C09063=1055.892,154.749,-84.853,171.715,33.030,156.169
C09064=1055.897,154.998,-84.876,171.717,33.033,156.169
C09065=1055.904,155.247,-84.898,171.719,33.035,156.170
C09066=1055.910,155.496,-84.919,171.720,33.038,156.170
C09067=1055.915,155.744,-84.942,171.722,33.041,156.170
C09068=1055.921,155.993,-84.963,171.724,33.043,156.171
C09069=1055.927,156.243,-84.985,171.726,33.045,156.171
C09070=1055.933,156.491,-85.008,171.728,33.048,156.172
C09071=1055.939,156.741,-85.030,171.730,33.050,156.172
C09072=1055.945,156.989,-85.051,171.732,33.053,156.173
C09073=1055.950,157.238,-85.074,171.734,33.055,156.173
C09074=1055.957,157.487,-85.096,171.736,33.058,156.173
C09075=1055.963,157.736,-85.117,171.738,33.061,156.174
C09076=1055.970,158.021,-85.143,171.740,33.064,156.174
C09077=1055.976,158.306,-85.168,171.742,33.066,156.175
C09078=1055.983,158.590,-85.193,171.745,33.070,156.175
C09079=1055.990,158.876,-85.218,171.747,33.072,156.176
C09080=1055.996,159.124,-85.241,171.749,33.075,156.176
C09081=1056.002,159.374,-85.263,171.751,33.077,156.177
C09082=1056.007,159.621,-85.285,171.753,33.080,156.177
C09083=1056.014,159.871,-85.307,171.755,33.082,156.178
C09084=1056.019,160.120,-85.330,171.757,33.085,156.178
C09085=1056.026,160.369,-85.351,171.758,33.087,156.178
C09086=1056.031,160.618,-85.374,171.760,33.090,156.179
C09087=1056.037,160.867,-85.396,171.762,33.093,156.179
C09088=1056.043,161.116,-85.419,171.764,33.095,156.180
C09089=1056.049,161.364,-85.440,171.766,33.098,156.180
C09090=1056.054,161.613,-85.463,171.768,33.100,156.181
C09091=1056.060,161.862,-85.486,171.770,33.103,156.181
C09092=1056.066,162.111,-85.508,171.772,33.106,156.182
C09093=1056.072,162.360,-85.530,171.774,33.109,156.182
C09094=1056.077,162.610,-85.553,171.776,33.111,156.182
C09095=1056.083,162.858,-85.575,171.778,33.114,156.183
C09096=1056.089,163.106,-85.598,171.780,33.116,156.183
C09097=1056.095,163.356,-85.620,171.782,33.119,156.184
C09098=1056.100,163.605,-85.643,171.784,33.122,156.184
C09099=1056.106,163.854,-85.666,171.786,33.125,156.185
C09100=1056.112,164.103,-85.687,171.788,33.127,156.185
C09101=1056.118,164.352,-85.710,171.790,33.130,156.186
C09102=1056.123,164.600,-85.733,171.792,33.132,156.186
C09103=1056.128,164.850,-85.755,171.794,33.135,156.186
C09104=1056.135,165.098,-85.778,171.796,33.137,156.187
C09105=1056.141,165.347,-85.800,171.798,33.141,156.187
C09106=1056.146,165.596,-85.823,171.800,33.143,156.188
C09107=1056.152,165.846,-85.846,171.802,33.146,156.188
C09108=1056.158,166.094,-85.868,171.804,33.148,156.189
C09109=1056.164,166.343,-85.891,171.806,33.151,156.189
C09110=1056.170,166.592,-85.914,171.807,33.153,156.190
C09111=1056.175,166.841,-85.936,171.809,33.156,156.190
C09112=1056.181,167.089,-85.958,171.811,33.159,156.191
C09113=1056.187,167.338,-85.981,171.813,33.162,156.191
C09114=1056.192,167.587,-86.004,171.815,33.164,156.192
C09115=1056.198,167.836,-86.027,171.817,33.167,156.192
C09116=1056.205,168.085,-86.049,171.819,33.169,156.192
C09117=1056.210,168.334,-86.072,171.821,33.172,156.193
C09118=1056.216,168.583,-86.094,171.823,33.175,156.193
C09119=1056.222,168.832,-86.117,171.825,33.178,156.194
C09120=1056.227,169.081,-86.140,171.827,33.180,156.194
C09121=1056.234,169.329,-86.163,171.829,33.183,156.195
C09122=1056.239,169.578,-86.186,171.832,33.185,156.195
C09123=1056.245,169.827,-86.209,171.834,33.188,156.196
C09124=1056.251,170.076,-86.232,171.836,33.190,156.196
C09125=1056.256,170.326,-86.254,171.838,33.194,156.197
C09126=1056.263,170.574,-86.276,171.840,33.196,156.197
C09127=1056.269,170.823,-86.299,171.842,33.199,156.197
C09128=1056.274,171.072,-86.322,171.844,33.201,156.198
C09129=1056.280,171.321,-86.345,171.847,33.204,156.198
C09130=1056.286,171.570,-86.368,171.849,33.206,156.199
C09131=1056.292,171.818,-86.390,171.851,33.210,156.199
C09132=1056.298,172.067,-86.413,171.853,33.212,156.200
C09133=1056.304,172.316,-86.436,171.855,33.215,156.200
C09134=1056.309,172.565,-86.459,171.857,33.217,156.201
C09135=1056.316,172.815,-86.482,171.859,33.220,156.201
C09136=1056.322,173.063,-86.505,171.861,33.222,156.202
C09137=1056.328,173.312,-86.528,171.863,33.225,156.202
C09138=1056.334,173.561,-86.551,171.865,33.228,156.203
C09139=1056.339,173.810,-86.574,171.867,33.231,156.203
C09140=1056.347,174.094,-86.600,171.869,33.234,156.204
C09141=1056.353,174.378,-86.626,171.872,33.236,156.204
C09142=1056.360,174.662,-86.653,171.874,33.240,156.204
C09143=1056.367,174.947,-86.678,171.876,33.243,156.205
C09144=1056.373,175.196,-86.701,171.879,33.245,156.205
C09145=1056.378,175.445,-86.724,171.881,33.248,156.206
C09146=1056.384,175.693,-86.747,171.883,33.250,156.206
C09147=1056.391,175.942,-86.771,171.885,33.253,156.207
C09148=1056.396,176.191,-86.794,171.887,33.256,156.207
C09149=1056.402,176.440,-86.817,171.889,33.259,156.208
C09150=1056.409,176.689,-86.839,171.891,33.261,156.208
C09151=1056.414,176.938,-86.862,171.893,33.264,156.209
C09152=1056.420,177.187,-86.885,171.895,33.266,156.209
C09153=1056.426,177.435,-86.909,171.897,33.269,156.210
C09154=1056.432,177.684,-86.932,171.899,33.271,156.210
C09155=1056.438,177.933,-86.955,171.901,33.275,156.211
C09156=1056.444,178.182,-86.978,171.904,33.277,156.211
C09157=1056.450,178.431,-87.001,171.906,33.280,156.211
C09158=1056.456,178.679,-87.024,171.908,33.282,156.212
C09159=1056.463,178.929,-87.048,171.910,33.285,156.212
C09160=1056.468,179.178,-87.070,171.912,33.287,156.213
C09161=1056.474,179.427,-87.093,171.914,33.291,156.213
C09162=1056.480,179.675,-87.117,171.916,33.293,156.214
C09163=1056.487,179.924,-87.140,171.918,33.296,156.214
C09164=1056.492,180.173,-87.163,171.920,33.298,156.215
C09165=1056.498,180.422,-87.187,171.923,33.301,156.215
C09166=1056.504,180.670,-87.210,171.925,33.304,156.216
C09167=1056.511,180.920,-87.233,171.927,33.307,156.216
C09168=1056.517,181.168,-87.256,171.929,33.309,156.216
C09169=1056.523,181.417,-87.279,171.931,33.312,156.217
C09170=1056.529,181.666,-87.302,171.933,33.314,156.217
C09171=1056.535,181.915,-87.326,171.935,33.317,156.218
C09172=1056.541,182.164,-87.349,171.937,33.320,156.218
C09173=1056.547,182.412,-87.373,171.940,33.323,156.219
C09174=1056.553,182.662,-87.396,171.942,33.325,156.219
C09175=1056.559,182.910,-87.419,171.944,33.328,156.220
C09176=1056.565,183.159,-87.443,171.946,33.330,156.220
C09177=1056.571,183.408,-87.466,171.948,33.333,156.221
C09178=1056.577,183.657,-87.490,171.950,33.336,156.221
C09179=1056.583,183.906,-87.513,171.952,33.338,156.222
C09180=1056.591,184.154,-87.536,171.955,33.341,156.222
C09181=1056.596,184.403,-87.560,171.957,33.344,156.222
C09182=1056.602,184.652,-87.583,171.959,33.347,156.223
C09183=1056.607,184.901,-87.606,171.961,33.349,156.223
C09184=1056.613,185.150,-87.631,171.963,33.352,156.224
C09185=1056.619,185.399,-87.654,171.965,33.355,156.224
C09186=1056.624,185.647,-87.678,171.967,33.358,156.225
C09187=1056.630,185.896,-87.702,171.970,33.361,156.225
C09188=1056.635,186.145,-87.725,171.972,33.364,156.226
C09189=1056.642,186.394,-87.749,171.974,33.366,156.226
C09190=1056.648,186.643,-87.772,171.977,33.370,156.227
C09191=1056.653,186.891,-87.797,171.979,33.372,156.227
C09192=1056.659,187.140,-87.820,171.981,33.375,156.228
C09193=1056.665,187.389,-87.844,171.983,33.378,156.228
C09194=1056.671,187.638,-87.868,171.986,33.381,156.229
C09195=1056.676,187.886,-87.892,171.988,33.384,156.229
C09196=1056.683,188.135,-87.916,171.990,33.387,156.230
C09197=1056.688,188.384,-87.939,171.992,33.389,156.230
C09198=1056.694,188.633,-87.963,171.994,33.392,156.231
C09199=1056.700,188.881,-87.987,171.996,33.395,156.231
C09200=1056.705,189.131,-88.011,171.998,33.398,156.232
C09201=1056.711,189.379,-88.034,172.001,33.401,156.232
C09202=1056.717,189.628,-88.059,172.003,33.404,156.233
C09203=1056.723,189.877,-88.083,172.005,33.406,156.233
C09204=1056.730,190.161,-88.110,172.007,33.409,156.234
C09205=1056.736,190.444,-88.137,172.010,33.413,156.235
C09206=1056.743,190.729,-88.164,172.012,33.416,156.235
C09207=1056.750,191.012,-88.192,172.015,33.420,156.236
C09208=1056.755,191.261,-88.215,172.017,33.422,156.236
C09209=1056.761,191.510,-88.240,172.019,33.425,156.237
C09210=1056.767,191.759,-88.263,172.021,33.428,156.237
C09211=1056.773,192.008,-88.288,172.024,33.431,156.238
C09212=1056.779,192.256,-88.312,172.026,33.433,156.238
C09213=1056.785,192.505,-88.336,172.028,33.437,156.239
C09214=1056.791,192.754,-88.360,172.030,33.439,156.239
C09215=1056.796,193.002,-88.384,172.032,33.442,156.240
C09216=1056.803,193.251,-88.408,172.035,33.445,156.240
C09217=1056.808,193.501,-88.432,172.037,33.448,156.241
C09218=1056.814,193.749,-88.455,172.039,33.451,156.241
C09219=1056.820,193.998,-88.480,172.041,33.454,156.242
C09220=1056.826,194.246,-88.504,172.044,33.456,156.242
C09221=1056.832,194.496,-88.528,172.047,33.459,156.243
C09222=1056.838,194.744,-88.552,172.049,33.462,156.243
C09223=1056.844,194.993,-88.577,172.051,33.465,156.244
C09224=1056.850,195.241,-88.600,172.053,33.468,156.244
C09225=1056.856,195.491,-88.625,172.056,33.471,156.245
C09226=1056.862,195.739,-88.649,172.058,33.474,156.245
C09227=1056.868,195.988,-88.673,172.060,33.476,156.246
C09228=1056.874,196.237,-88.697,172.062,33.480,156.246
C09229=1056.880,196.486,-88.721,172.065,33.482,156.247
C09230=1056.886,196.734,-88.746,172.067,33.485,156.247
C09231=1056.892,196.983,-88.770,172.069,33.488,156.248
C09232=1056.897,197.231,-88.795,172.071,33.491,156.248
C09233=1056.904,197.480,-88.819,172.074,33.494,156.249
C09234=1056.909,197.729,-88.843,172.076,33.497,156.249
C09235=1056.916,197.978,-88.867,172.078,33.500,156.250
C09236=1056.921,198.227,-88.891,172.080,33.502,156.250
C09237=1056.928,198.476,-88.915,172.083,33.506,156.251
C09238=1056.933,198.724,-88.940,172.085,33.508,156.251
C09239=1056.940,198.972,-88.964,172.087,33.511,156.252
C09240=1056.945,199.221,-88.989,172.090,33.514,156.252
C09241=1056.952,199.470,-89.013,172.092,33.517,156.253
C09242=1056.958,199.719,-89.037,172.094,33.520,156.253
C09243=1056.963,199.968,-89.061,172.096,33.523,156.254
C09244=1056.970,200.216,-89.086,172.099,33.526,156.254
C09245=1056.975,200.465,-89.110,172.101,33.528,156.255
C09246=1056.982,200.714,-89.135,172.104,33.531,156.255
C09247=1056.988,200.963,-89.159,172.107,33.535,156.256
C09248=1056.994,201.211,-89.183,172.109,33.537,156.256
C09249=1057.000,201.460,-89.208,172.111,33.540,156.257
C09250=1057.005,201.709,-89.232,172.113,33.543,156.257
C09251=1057.012,201.957,-89.257,172.116,33.546,156.258
C09252=1057.018,202.206,-89.282,172.118,33.549,156.259
C09253=1057.024,202.455,-89.306,172.120,33.552,156.259
C09254=1057.030,202.704,-89.331,172.123,33.555,156.260
C09255=1057.035,202.952,-89.356,172.125,33.558,156.260
C09256=1057.041,203.201,-89.380,172.127,33.561,156.261
C09257=1057.047,203.450,-89.406,172.130,33.564,156.261
C09258=1057.053,203.698,-89.429,172.132,33.567,156.262
C09259=1057.059,203.947,-89.455,172.134,33.570,156.262
C09260=1057.065,204.196,-89.479,172.136,33.573,156.263
C09261=1057.071,204.444,-89.504,172.139,33.576,156.263
C09262=1057.077,204.694,-89.529,172.141,33.579,156.264
C09263=1057.082,204.942,-89.554,172.143,33.582,156.264
C09264=1057.088,205.191,-89.578,172.146,33.585,156.265
C09265=1057.095,205.440,-89.604,172.148,33.588,156.266
C09266=1057.101,205.688,-89.627,172.151,33.591,156.266
C09267=1057.107,205.936,-89.653,172.154,33.594,156.267
C09268=1057.131,206.987,-89.757,172.349,33.683,156.279
C09269=1057.138,207.224,-89.781,172.351,33.687,156.279
C09270=1057.144,207.459,-89.806,172.353,33.690,156.280
C09271=1057.150,207.696,-89.831,172.354,33.694,156.281
C09272=1057.156,207.931,-89.855,172.356,33.698,156.282
C09273=1057.162,208.168,-89.879,172.358,33.702,156.282
C09274=1057.167,208.404,-89.904,172.360,33.705,156.283
C09275=1057.173,208.640,-89.929,172.361,33.709,156.284
C09276=1057.179,208.875,-89.953,172.363,33.713,156.284
C09277=1057.185,209.124,-89.979,172.365,33.716,156.285
C09278=1057.191,209.372,-90.005,172.368,33.720,156.286
C09279=1057.198,209.622,-90.031,172.370,33.724,156.287
C09280=1057.204,209.870,-90.057,172.371,33.728,156.287
C09281=1057.210,210.119,-90.083,172.373,33.731,156.288
C09282=1057.216,210.367,-90.109,172.375,33.736,156.289
C09283=1057.223,210.615,-90.134,172.377,33.739,156.289
C09284=1057.228,210.864,-90.161,172.379,33.744,156.290
C09285=1057.235,211.113,-90.186,172.381,33.747,156.291
C09286=1057.242,211.361,-90.212,172.383,33.751,156.292
C09287=1057.247,211.610,-90.238,172.385,33.755,156.293
C09288=1057.254,211.858,-90.264,172.387,33.759,156.293
C09289=1057.260,212.107,-90.290,172.389,33.762,156.294
C09290=1057.266,212.355,-90.316,172.391,33.767,156.295
C09291=1057.272,212.605,-90.342,172.393,33.770,156.295
C09292=1057.278,212.853,-90.369,172.395,33.774,156.296
C09293=1057.284,213.102,-90.394,172.397,33.778,156.297
C09294=1057.290,213.350,-90.421,172.399,33.782,156.298
C09295=1057.297,213.598,-90.447,172.400,33.785,156.298
C09296=1057.303,213.848,-90.473,172.402,33.790,156.299
C09297=1057.309,214.096,-90.499,172.405,33.793,156.300
C09298=1057.315,214.344,-90.526,172.407,33.797,156.301
C09299=1057.321,214.593,-90.551,172.409,33.801,156.301
C09300=1057.327,214.841,-90.578,172.411,33.805,156.302
C09301=1057.334,215.090,-90.604,172.413,33.809,156.303
C09302=1057.340,215.339,-90.630,172.415,33.813,156.304
C09303=1057.346,215.587,-90.656,172.417,33.817,156.304
C09304=1057.352,215.835,-90.683,172.419,33.820,156.305
C09305=1057.359,216.084,-90.709,172.421,33.824,156.306
C09306=1057.365,216.333,-90.735,172.423,33.828,156.306
C09307=1057.371,216.581,-90.761,172.425,33.832,156.307
C09308=1057.377,216.829,-90.788,172.427,33.836,156.308
C09309=1057.384,217.078,-90.814,172.429,33.840,156.309
C09310=1057.389,217.327,-90.840,172.431,33.843,156.309
C09311=1057.396,217.575,-90.866,172.433,33.847,156.310
C09312=1057.402,217.824,-90.893,172.435,33.851,156.311
C09313=1057.408,218.073,-90.920,172.437,33.855,156.312
C09314=1057.415,218.321,-90.946,172.440,33.858,156.312
C09315=1057.420,218.570,-90.972,172.442,33.863,156.313
C09316=1057.427,218.818,-90.998,172.444,33.866,156.314
C09317=1057.433,219.067,-91.025,172.446,33.870,156.314
C09318=1057.439,219.315,-91.051,172.448,33.874,156.315
C09319=1057.446,219.564,-91.078,172.449,33.877,156.316
C09320=1057.452,219.812,-91.104,172.451,33.881,156.317
C09321=1057.458,220.060,-91.131,172.453,33.885,156.317
C09322=1057.464,220.309,-91.158,172.456,33.889,156.318
C09323=1057.471,220.557,-91.184,172.458,33.892,156.319
C09324=1057.477,220.806,-91.211,172.460,33.897,156.320
C09325=1057.483,221.045,-91.236,172.462,33.900,156.320
C09326=1057.489,221.284,-91.261,172.464,33.904,156.321
C09327=1057.495,221.522,-91.287,172.466,33.907,156.322
C09328=1057.501,221.761,-91.312,172.468,33.911,156.322
C09329=1057.506,222.000,-91.338,172.470,33.915,156.323
C09330=1057.512,222.238,-91.364,172.473,33.918,156.324
C09331=1057.519,222.477,-91.389,172.474,33.922,156.325
C09332=1057.525,222.715,-91.415,172.476,33.926,156.325
C09333=1057.531,222.964,-91.442,172.478,33.929,156.326
C09334=1057.536,223.212,-91.468,172.480,33.933,156.327
C09335=1057.543,223.461,-91.495,172.482,33.937,156.327
C09336=1057.549,223.709,-91.522,172.484,33.941,156.328
C09337=1057.555,223.957,-91.548,172.486,33.944,156.329
C09338=1057.562,224.206,-91.575,172.489,33.948,156.330
C09339=1057.567,224.455,-91.602,172.491,33.952,156.330
C09340=1057.574,224.703,-91.629,172.493,33.956,156.331
C09341=1057.580,224.952,-91.656,172.495,33.960,156.332
C09342=1057.586,225.200,-91.683,172.497,33.963,156.332
C09343=1057.593,225.449,-91.709,172.499,33.967,156.333
C09344=1057.598,225.697,-91.736,172.501,33.971,156.334
C09345=1057.605,225.946,-91.763,172.503,33.975,156.335
C09346=1057.611,226.194,-91.790,172.506,33.978,156.335
C09347=1057.617,226.443,-91.817,172.508,33.982,156.336
C09348=1057.623,226.691,-91.844,172.510,33.986,156.337
C09349=1057.630,226.940,-91.870,172.512,33.990,156.338
C09350=1057.636,227.188,-91.898,172.514,33.994,156.338
C09351=1057.643,227.437,-91.925,172.516,33.997,156.339
C09352=1057.648,227.685,-91.951,172.518,34.001,156.340
C09353=1057.654,227.934,-91.978,172.521,34.005,156.341
C09354=1057.661,228.182,-92.006,172.523,34.009,156.341
C09355=1057.667,228.431,-92.033,172.525,34.012,156.342
C09356=1057.674,228.679,-92.059,172.527,34.016,156.343
C09357=1057.680,228.928,-92.086,172.529,34.020,156.343
C09358=1057.686,229.176,-92.113,172.532,34.023,156.344
C09359=1057.693,229.425,-92.140,172.534,34.027,156.345
C09360=1057.699,229.673,-92.167,172.537,34.031,156.346
C09361=1057.705,229.922,-92.195,172.539,34.035,156.346
C09362=1057.711,230.170,-92.222,172.541,34.038,156.347
C09363=1057.717,230.419,-92.249,172.543,34.042,156.348
C09364=1057.724,230.666,-92.276,172.545,34.046,156.348
C09365=1057.730,230.915,-92.303,172.547,34.050,156.349
C09366=1057.735,231.164,-92.331,172.549,34.054,156.350
C09367=1057.742,231.413,-92.358,172.552,34.057,156.351
C09368=1057.747,231.661,-92.385,172.554,34.061,156.351
C09369=1057.754,231.909,-92.413,172.556,34.065,156.352
C09370=1057.760,232.158,-92.439,172.558,34.069,156.353
C09371=1057.767,232.406,-92.467,172.560,34.072,156.354
C09372=1057.773,232.654,-92.494,172.562,34.076,156.354
C09373=1057.779,232.903,-92.521,172.564,34.080,156.355
C09374=1057.786,233.151,-92.549,172.567,34.084,156.356
C09375=1057.791,233.400,-92.576,172.569,34.087,156.356
C09376=1057.797,233.648,-92.604,172.572,34.091,156.357
C09377=1057.803,233.897,-92.631,172.574,34.095,156.358
C09378=1057.810,234.145,-92.658,172.576,34.099,156.359
C09379=1057.816,234.393,-92.686,172.578,34.103,156.359
C09380=1057.822,234.642,-92.713,172.580,34.106,156.360
C09381=1057.827,234.877,-92.739,172.583,34.110,156.361
C09382=1057.833,235.112,-92.765,172.585,34.113,156.361
C09383=1057.840,235.346,-92.791,172.587,34.117,156.362
C09384=1057.845,235.581,-92.818,172.589,34.121,156.363
C09385=1057.851,235.815,-92.843,172.591,34.124,156.363
C09386=1057.857,236.050,-92.869,172.593,34.127,156.364
C09387=1057.863,236.285,-92.895,172.595,34.131,156.365
C09388=1057.868,236.520,-92.921,172.598,34.135,156.366
C09389=1057.875,236.768,-92.949,172.600,34.138,156.366
C09390=1057.881,237.016,-92.977,172.602,34.142,156.367
C09391=1057.887,237.264,-93.004,172.604,34.145,156.368
C09392=1057.893,237.514,-93.032,172.606,34.150,156.369
C09393=1057.900,237.762,-93.059,172.608,34.153,156.369
C09394=1057.906,238.010,-93.087,172.611,34.157,156.370
C09395=1057.912,238.258,-93.114,172.614,34.161,156.371
C09396=1057.918,238.507,-93.143,172.616,34.164,156.371
C09397=1057.924,238.755,-93.169,172.618,34.168,156.372
C09398=1057.931,239.004,-93.197,172.620,34.172,156.373
C09399=1057.938,239.252,-93.225,172.622,34.176,156.374
C09400=1057.943,239.500,-93.253,172.624,34.179,156.374
C09401=1057.950,239.749,-93.281,172.627,34.183,156.375
C09402=1057.956,239.997,-93.308,172.629,34.186,156.376
C09403=1057.962,240.246,-93.337,172.632,34.190,156.376
C09404=1057.968,240.494,-93.364,172.634,34.194,156.377
C09405=1057.975,240.742,-93.392,172.636,34.198,156.378
C09406=1057.981,240.991,-93.419,172.638,34.202,156.379
C09407=1057.987,241.240,-93.447,172.641,34.205,156.379
C09408=1057.993,241.488,-93.474,172.643,34.209,156.380
C09409=1057.999,241.736,-93.503,172.646,34.212,156.381
C09410=1058.006,241.985,-93.530,172.648,34.216,156.381
C09411=1058.012,242.234,-93.559,172.650,34.220,156.382
C09412=1058.018,242.481,-93.586,172.652,34.224,156.383
C09413=1058.024,242.729,-93.615,172.655,34.228,156.384
C09414=1058.031,242.978,-93.643,172.657,34.231,156.384
C09415=1058.036,243.226,-93.671,172.660,34.235,156.385
C09416=1058.043,243.474,-93.699,172.662,34.238,156.386
C09417=1058.049,243.723,-93.727,172.664,34.243,156.387
C09418=1058.056,243.972,-93.755,172.666,34.246,156.387
C09419=1058.061,244.220,-93.783,172.669,34.250,156.388
C09420=1058.067,244.468,-93.811,172.671,34.253,156.389
C09421=1058.074,244.716,-93.839,172.674,34.257,156.389
C09422=1058.080,244.965,-93.868,172.676,34.261,156.390
C09423=1058.086,245.213,-93.895,172.678,34.265,156.391
C09424=1058.092,245.461,-93.923,172.680,34.269,156.392
C09425=1058.098,245.710,-93.952,172.683,34.272,156.392
C09426=1058.104,245.959,-93.979,172.686,34.276,156.393
C09427=1058.111,246.207,-94.008,172.688,34.279,156.394
C09428=1058.117,246.455,-94.036,172.690,34.284,156.395
C09429=1058.123,246.703,-94.064,172.692,34.287,156.395
C09430=1058.129,246.951,-94.093,172.694,34.291,156.396
C09431=1058.135,247.200,-94.122,172.698,34.295,156.397
C09432=1058.141,247.449,-94.150,172.700,34.299,156.398
C09433=1058.147,247.696,-94.178,172.702,34.302,156.398
C09434=1058.153,247.945,-94.206,172.704,34.306,156.399
C09435=1058.159,248.193,-94.235,172.706,34.310,156.400
C09436=1058.165,248.442,-94.264,172.710,34.314,156.401
C09437=1058.171,248.674,-94.290,172.712,34.317,156.401
C09438=1058.177,248.905,-94.316,172.714,34.320,156.402
C09439=1058.182,249.137,-94.343,172.716,34.324,156.403
C09440=1058.188,249.369,-94.369,172.718,34.328,156.403
C09441=1058.193,249.600,-94.397,172.720,34.331,156.404
C09442=1058.200,249.831,-94.422,172.723,34.335,156.405
C09443=1058.205,250.063,-94.449,172.725,34.338,156.405
C09444=1058.211,250.295,-94.476,172.727,34.341,156.406
C09445=1058.217,250.544,-94.504,172.730,34.346,156.407
C09446=1058.224,250.791,-94.533,172.732,34.349,156.408
C09447=1058.229,251.040,-94.561,172.734,34.353,156.408
C09448=1058.235,251.288,-94.590,172.737,34.356,156.409
C09449=1058.241,251.536,-94.618,172.740,34.360,156.410
C09450=1058.247,251.784,-94.647,172.742,34.364,156.410
C09451=1058.253,252.033,-94.675,172.744,34.368,156.411
C09452=1058.260,252.281,-94.704,172.746,34.371,156.412
C09453=1058.266,252.529,-94.733,172.750,34.375,156.413
C09454=1058.272,252.778,-94.761,172.752,34.379,156.413
C09455=1058.279,253.026,-94.790,172.754,34.383,156.414
C09456=1058.285,253.275,-94.819,172.756,34.387,156.415
C09457=1058.291,253.523,-94.848,172.759,34.390,156.416
C09458=1058.297,253.771,-94.877,172.762,34.394,156.416
C09459=1058.303,254.020,-94.905,172.764,34.397,156.417
C09460=1058.310,254.268,-94.933,172.767,34.401,156.418
C09461=1058.316,254.516,-94.963,172.769,34.405,156.419
C09462=1058.322,254.764,-94.991,172.771,34.409,156.419
C09463=1058.328,255.013,-95.020,172.773,34.412,156.420
C09464=1058.335,255.261,-95.049,172.777,34.416,156.421
C09465=1058.341,255.509,-95.078,172.779,34.420,156.421
C09466=1058.347,255.758,-95.106,172.781,34.423,156.422
C09467=1058.353,256.006,-95.135,172.784,34.427,156.423
C09468=1058.359,256.254,-95.164,172.786,34.431,156.424
C09469=1058.366,256.502,-95.193,172.789,34.435,156.424
C09470=1058.372,256.750,-95.221,172.792,34.438,156.425
C09471=1058.379,256.999,-95.250,172.794,34.442,156.426
C09472=1058.385,257.247,-95.279,172.796,34.445,156.426
C09473=1058.391,257.495,-95.308,172.799,34.449,156.427
C09474=1058.397,257.743,-95.337,172.802,34.453,156.428
C09475=1058.404,257.991,-95.366,172.804,34.457,156.429
C09476=1058.410,258.240,-95.395,172.807,34.460,156.429
C09477=1058.416,258.488,-95.424,172.809,34.464,156.430
C09478=1058.422,258.736,-95.453,172.811,34.468,156.431
C09479=1058.428,258.984,-95.482,172.815,34.471,156.432
C09480=1058.435,259.232,-95.511,172.817,34.475,156.432
C09481=1058.441,259.481,-95.540,172.819,34.478,156.433
C09482=1058.448,259.729,-95.569,172.822,34.483,156.434
C09483=1058.455,259.977,-95.598,172.824,34.486,156.435
C09484=1058.461,260.225,-95.627,172.827,34.490,156.435
C09485=1058.467,260.473,-95.656,172.830,34.494,156.436
C09486=1058.473,260.722,-95.685,172.832,34.497,156.437
C09487=1058.480,260.970,-95.714,172.835,34.501,156.437
C09488=1058.486,261.219,-95.743,172.837,34.504,156.438
C09489=1058.493,261.467,-95.772,172.840,34.508,156.439
C09490=1058.499,261.715,-95.801,172.843,34.512,156.440
C09491=1058.505,261.963,-95.830,172.845,34.515,156.440
C09492=1058.511,262.211,-95.859,172.848,34.519,156.441
C09493=1058.517,262.442,-95.887,172.850,34.522,156.442
C09494=1058.524,262.673,-95.914,172.853,34.526,156.442
C09495=1058.529,262.903,-95.941,172.855,34.529,156.443
C09496=1058.536,263.134,-95.968,172.857,34.532,156.444
C09497=1058.541,263.365,-95.995,172.860,34.536,156.444
C09498=1058.547,263.595,-96.023,172.862,34.540,156.445
C09499=1058.553,263.826,-96.050,172.864,34.543,156.446
C09500=1058.558,264.057,-96.078,172.867,34.546,156.446
C09501=1058.565,264.305,-96.107,172.870,34.550,156.447
C09502=1058.571,264.553,-96.136,172.872,34.554,156.448
C09503=1058.577,264.801,-96.165,172.875,34.558,156.449
C09504=1058.583,265.049,-96.195,172.877,34.561,156.449
C09505=1058.589,265.297,-96.225,172.880,34.565,156.450
C09506=1058.596,265.546,-96.254,172.883,34.569,156.451
C09507=1058.602,265.794,-96.284,172.885,34.573,156.452
C09508=1058.608,266.042,-96.314,172.888,34.576,156.452
C09509=1058.615,266.290,-96.343,172.891,34.580,156.453
C09510=1058.620,266.538,-96.372,172.893,34.584,156.454
C09511=1058.627,266.786,-96.402,172.896,34.588,156.455
C09512=1058.634,267.035,-96.431,172.898,34.591,156.455
C09513=1058.639,267.283,-96.461,172.901,34.595,156.456
C09514=1058.646,267.531,-96.491,172.904,34.599,156.457
C09515=1058.652,267.779,-96.520,172.907,34.603,156.458
C09516=1058.658,268.027,-96.551,172.909,34.606,156.458
C09517=1058.665,268.275,-96.580,172.911,34.610,156.459
C09518=1058.671,268.523,-96.609,172.914,34.613,156.460
C09519=1058.677,268.772,-96.639,172.917,34.617,156.461
C09520=1058.683,269.020,-96.668,172.920,34.621,156.461
C09521=1058.689,269.268,-96.699,172.922,34.625,156.462
C09522=1058.695,269.516,-96.728,172.925,34.628,156.463
C09523=1058.702,269.765,-96.758,172.928,34.632,156.464
C09524=1058.708,270.012,-96.788,172.931,34.636,156.464
C09525=1058.714,270.261,-96.818,172.933,34.640,156.465
C09526=1058.721,270.509,-96.848,172.936,34.644,156.466
C09527=1058.727,270.757,-96.878,172.939,34.647,156.467
C09528=1058.733,271.005,-96.907,172.942,34.651,156.467
C09529=1058.740,271.253,-96.938,172.944,34.655,156.468
C09530=1058.746,271.501,-96.967,172.946,34.659,156.469
C09531=1058.752,271.749,-96.998,172.949,34.662,156.470
C09532=1058.759,271.998,-97.027,172.952,34.666,156.470
C09533=1058.764,272.246,-97.057,172.955,34.670,156.471
C09534=1058.771,272.493,-97.087,172.957,34.674,156.472
C09535=1058.777,272.742,-97.118,172.960,34.677,156.473
C09536=1058.784,272.990,-97.147,172.963,34.681,156.473
C09537=1058.789,273.238,-97.177,172.966,34.685,156.474
C09538=1058.796,273.486,-97.208,172.968,34.689,156.475
C09539=1058.802,273.734,-97.238,172.971,34.692,156.476
C09540=1058.808,273.982,-97.267,172.974,34.696,156.476
C09541=1058.815,274.231,-97.297,172.977,34.700,156.477
C09542=1058.821,274.478,-97.328,172.979,34.703,156.478
C09543=1058.827,274.726,-97.358,172.982,34.708,156.479
C09544=1058.834,274.974,-97.388,172.984,34.711,156.479
C09545=1058.839,275.223,-97.418,172.988,34.715,156.480
C09546=1058.846,275.471,-97.449,172.990,34.719,156.481
C09547=1058.852,275.719,-97.478,172.993,34.723,156.482
C09548=1058.858,275.967,-97.509,172.995,34.726,156.482
C09549=1058.864,276.200,-97.537,172.999,34.730,156.483
C09550=1058.870,276.432,-97.565,173.001,34.733,156.484
C09551=1058.876,276.665,-97.594,173.004,34.737,156.485
C09552=1058.882,276.897,-97.622,173.006,34.740,156.485
C09553=1058.888,277.130,-97.651,173.009,34.744,156.486
C09554=1058.893,277.362,-97.679,173.012,34.748,156.487
C09555=1058.900,277.595,-97.708,173.014,34.751,156.488
C09556=1058.905,277.827,-97.736,173.016,34.755,156.488
C09557=1058.912,278.076,-97.767,173.019,34.758,156.489
C09558=1058.918,278.324,-97.797,173.023,34.762,156.490
C09559=1058.924,278.572,-97.828,173.025,34.766,156.491
C09560=1058.931,278.820,-97.858,173.028,34.770,156.491
C09561=1058.937,279.068,-97.889,173.030,34.774,156.492
C09562=1058.943,279.316,-97.919,173.034,34.777,156.493
C09563=1058.949,279.564,-97.950,173.036,34.781,156.494
C09564=1058.956,279.812,-97.979,173.039,34.785,156.494
C09565=1058.962,280.060,-98.010,173.042,34.789,156.495
C09566=1058.968,280.308,-98.041,173.045,34.792,156.496
C09567=1058.975,280.556,-98.072,173.048,34.796,156.497
C09568=1058.981,280.804,-98.102,173.050,34.800,156.497
C09569=1058.987,281.053,-98.133,173.053,34.804,156.498
C09570=1058.993,281.300,-98.164,173.056,34.808,156.499
C09571=1059.000,281.548,-98.195,173.059,34.812,156.500
C09572=1059.005,281.796,-98.225,173.062,34.815,156.501
C09573=1059.012,282.045,-98.256,173.064,34.820,156.501
C09574=1059.018,282.292,-98.287,173.068,34.823,156.502
C09575=1059.024,282.540,-98.318,173.070,34.827,156.503
C09576=1059.030,282.788,-98.348,173.073,34.831,156.504
C09577=1059.037,283.036,-98.379,173.076,34.834,156.504
C09578=1059.043,283.284,-98.410,173.079,34.839,156.505
C09579=1059.049,283.532,-98.440,173.082,34.842,156.506
C09580=1059.056,283.780,-98.472,173.084,34.846,156.507
C09581=1059.062,284.028,-98.502,173.088,34.850,156.508
C09582=1059.068,284.277,-98.533,173.091,34.854,156.508
C09583=1059.074,284.524,-98.564,173.093,34.858,156.509
C09584=1059.081,284.772,-98.595,173.096,34.862,156.510
C09585=1059.087,285.020,-98.626,173.100,34.865,156.511
C09586=1059.093,285.268,-98.657,173.102,34.869,156.512
C09587=1059.100,285.516,-98.688,173.105,34.873,156.512
C09588=1059.106,285.764,-98.718,173.107,34.877,156.513
C09589=1059.112,286.012,-98.750,173.111,34.881,156.514
C09590=1059.119,286.260,-98.780,173.114,34.884,156.515
C09591=1059.125,286.507,-98.812,173.116,34.888,156.515
C09592=1059.131,286.756,-98.842,173.119,34.892,156.516
C09593=1059.138,287.004,-98.874,173.123,34.896,156.517
C09594=1059.144,287.252,-98.904,173.125,34.900,156.518
C09595=1059.151,287.500,-98.935,173.128,34.904,156.519
C09596=1059.157,287.748,-98.967,173.131,34.907,156.519
C09597=1059.162,287.996,-98.998,173.134,34.911,156.520
C09598=1059.169,288.244,-99.029,173.137,34.915,156.521
C09599=1059.176,288.492,-99.060,173.140,34.919,156.522
C09600=1059.182,288.740,-99.091,173.143,34.923,156.522
C09601=1059.188,288.987,-99.123,173.146,34.927,156.523
C09602=1059.195,289.235,-99.154,173.149,34.930,156.524
C09603=1059.201,289.484,-99.185,173.151,34.935,156.525
C09604=1059.207,289.731,-99.216,173.155,34.938,156.526
C09605=1059.213,289.969,-99.246,173.158,34.942,156.526
C09606=1059.219,290.207,-99.276,173.160,34.946,156.527
C09607=1059.225,290.445,-99.307,173.163,34.949,156.528
C09608=1059.231,290.683,-99.336,173.166,34.953,156.529
C09609=1059.237,290.921,-99.367,173.169,34.957,156.529
C09610=1059.244,291.160,-99.397,173.172,34.961,156.530
C09611=1059.250,291.398,-99.427,173.175,34.965,156.531
C09612=1059.255,291.636,-99.457,173.178,34.968,156.532
C09613=1059.262,291.884,-99.489,173.181,34.972,156.533
C09614=1059.268,292.131,-99.520,173.183,34.976,156.533
C09615=1059.274,292.379,-99.552,173.187,34.980,156.534
C09616=1059.281,292.627,-99.583,173.190,34.984,156.535
C09617=1059.288,292.875,-99.615,173.192,34.988,156.536
C09618=1059.293,293.123,-99.646,173.196,34.992,156.537
C09619=1059.300,293.370,-99.678,173.199,34.995,156.537
C09620=1059.306,293.618,-99.709,173.202,35.000,156.538
C09621=1059.312,293.867,-99.741,173.204,35.003,156.539
C09622=1059.319,294.114,-99.773,173.208,35.007,156.540
C09623=1059.325,294.362,-99.804,173.211,35.011,156.541
C09624=1059.331,294.610,-99.836,173.214,35.015,156.541
C09625=1059.338,294.858,-99.867,173.217,35.019,156.542
C09626=1059.345,295.106,-99.899,173.220,35.023,156.543
C09627=1059.351,295.354,-99.931,173.223,35.027,156.544
C09628=1059.357,295.602,-99.962,173.226,35.031,156.545
C09629=1059.363,295.849,-99.994,173.229,35.035,156.545
C09630=1059.370,296.097,-100.026,173.232,35.039,156.546
C09631=1059.376,296.345,-100.058,173.235,35.043,156.547
C09632=1059.382,296.593,-100.089,173.239,35.047,156.548
C09633=1059.388,296.841,-100.121,173.241,35.050,156.549
C09634=1059.394,297.089,-100.153,173.244,35.054,156.550
C09635=1059.401,297.336,-100.185,173.248,35.059,156.550
C09636=1059.407,297.584,-100.217,173.251,35.063,156.551
C09637=1059.413,297.832,-100.249,173.253,35.067,156.552
C09638=1059.420,298.079,-100.281,173.257,35.071,156.553
C09639=1059.426,298.328,-100.313,173.260,35.075,156.554
C09640=1059.432,298.576,-100.345,173.263,35.079,156.555
C09641=1059.438,298.823,-100.378,173.266,35.083,156.555
C09642=1059.444,299.071,-100.410,173.269,35.087,156.556
C09643=1059.450,299.319,-100.441,173.272,35.091,156.557
C09644=1059.457,299.566,-100.474,173.275,35.095,156.558
C09645=1059.463,299.815,-100.506,173.279,35.099,156.559
C09646=1059.469,300.062,-100.539,173.281,35.103,156.560
C09647=1059.476,300.310,-100.570,173.284,35.107,156.561
C09648=1059.482,300.558,-100.603,173.288,35.111,156.561
C09649=1059.488,300.806,-100.635,173.291,35.115,156.562
C09650=1059.494,301.054,-100.668,173.294,35.119,156.563
C09651=1059.501,301.301,-100.699,173.298,35.123,156.564
C09652=1059.507,301.549,-100.732,173.300,35.127,156.565
C09653=1059.513,301.797,-100.764,173.303,35.131,156.566
C09654=1059.519,302.045,-100.797,173.307,35.136,156.566
C09655=1059.525,302.293,-100.829,173.310,35.140,156.567
C09656=1059.532,302.541,-100.861,173.313,35.144,156.568
C09657=1059.538,302.787,-100.893,173.317,35.148,156.569
C09658=1059.544,303.035,-100.925,173.319,35.151,156.570
C09659=1059.550,303.283,-100.958,173.322,35.155,156.571
C09660=1059.557,303.532,-100.990,173.326,35.160,156.571
C09661=1059.563,303.777,-101.022,173.329,35.164,156.572
C09662=1059.569,304.022,-101.055,173.332,35.168,156.573
C09663=1059.576,304.268,-101.087,173.336,35.172,156.574
C09664=1059.582,304.514,-101.119,173.338,35.176,156.575
C09665=1059.589,304.760,-101.151,173.341,35.180,156.576
C09666=1059.595,305.005,-101.183,173.345,35.184,156.577
C09667=1059.601,305.251,-101.216,173.348,35.188,156.577
C09668=1059.608,305.497,-101.248,173.351,35.192,156.578
C09669=1059.614,305.744,-101.281,173.355,35.196,156.579
C09670=1059.620,305.992,-101.313,173.358,35.200,156.580
C09671=1059.626,306.240,-101.345,173.361,35.204,156.581
C09672=1059.633,306.488,-101.378,173.364,35.208,156.582
C09673=1059.640,306.735,-101.411,173.367,35.212,156.582
C09674=1059.646,306.983,-101.443,173.370,35.216,156.583
C09675=1059.653,307.231,-101.476,173.374,35.221,156.584
C09676=1059.659,307.478,-101.509,173.377,35.225,156.585
C09677=1059.665,307.726,-101.541,173.380,35.229,156.586
C09678=1059.671,307.974,-101.574,173.384,35.233,156.587
C09679=1059.678,308.222,-101.607,173.387,35.237,156.588
C09680=1059.684,308.470,-101.639,173.390,35.241,156.588
C09681=1059.691,308.718,-101.672,173.394,35.245,156.589
C09682=1059.698,308.965,-101.704,173.397,35.249,156.590
C09683=1059.704,309.212,-101.737,173.400,35.253,156.591
C09684=1059.711,309.461,-101.770,173.404,35.257,156.592
C09685=1059.717,309.708,-101.803,173.407,35.262,156.593
C09686=1059.724,309.956,-101.836,173.409,35.266,156.594
C09687=1059.730,310.203,-101.868,173.413,35.270,156.595
C09688=1059.737,310.452,-101.901,173.416,35.274,156.595
C09689=1059.743,310.699,-101.934,173.419,35.278,156.596
C09690=1059.750,310.946,-101.968,173.423,35.282,156.597
C09691=1059.757,311.195,-102.001,173.426,35.286,156.598
C09692=1059.763,311.442,-102.034,173.429,35.290,156.599
C09693=1059.769,311.690,-102.066,173.433,35.294,156.600
C09694=1059.776,311.937,-102.098,173.436,35.298,156.601
C09695=1059.783,312.185,-102.132,173.440,35.302,156.601
C09696=1059.789,312.433,-102.164,173.443,35.306,156.602
C09697=1059.797,312.681,-102.198,173.446,35.311,156.603
C09698=1059.803,312.928,-102.231,173.450,35.315,156.604
C09699=1059.809,313.176,-102.264,173.453,35.319,156.605
C09700=1059.816,313.424,-102.297,173.456,35.323,156.606
C09701=1059.823,313.671,-102.330,173.460,35.327,156.607
C09702=1059.828,313.919,-102.363,173.463,35.332,156.608
C09703=1059.835,314.167,-102.397,173.466,35.336,156.608
C09704=1059.842,314.414,-102.430,173.470,35.340,156.609
C09705=1059.847,314.662,-102.463,173.473,35.344,156.610
C09706=1059.854,314.909,-102.497,173.477,35.349,156.611
C09707=1059.860,315.158,-102.531,173.480,35.353,156.612
C09708=1059.867,315.405,-102.564,173.483,35.357,156.613
C09709=1059.872,315.653,-102.597,173.487,35.362,156.614
C09710=1059.879,315.900,-102.631,173.490,35.366,156.615
C09711=1059.885,316.148,-102.665,173.494,35.370,156.616
C09712=1059.891,316.395,-102.698,173.497,35.375,156.617
C09713=1059.898,316.644,-102.732,173.500,35.379,156.618
C09714=1059.904,316.891,-102.765,173.504,35.383,156.619
C09715=1059.910,317.139,-102.798,173.507,35.387,156.620
C09716=1059.917,317.386,-102.832,173.510,35.392,156.620
C09717=1059.923,317.634,-102.866,173.514,35.396,156.621
C09718=1059.930,317.882,-102.899,173.517,35.401,156.622
C09719=1059.936,318.129,-102.933,173.521,35.405,156.623
C09720=1059.942,318.377,-102.966,173.524,35.409,156.624
C09721=1059.948,318.625,-103.001,173.527,35.413,156.625
C09722=1059.955,318.872,-103.034,173.531,35.418,156.626
C09723=1059.961,319.120,-103.069,173.534,35.422,156.627
C09724=1059.968,319.367,-103.101,173.538,35.426,156.628
C09725=1059.974,319.615,-103.136,173.541,35.431,156.629
C09726=1059.981,319.862,-103.169,173.545,35.435,156.630
C09727=1059.987,320.110,-103.204,173.549,35.440,156.631
C09728=1059.994,320.358,-103.236,173.552,35.444,156.632
C09729=1060.000,320.606,-103.271,173.556,35.448,156.633
C09730=1060.007,320.853,-103.304,173.559,35.452,156.633
C09731=1060.013,321.101,-103.339,173.562,35.457,156.634
C09732=1060.020,321.348,-103.372,173.566,35.461,156.635
C09733=1060.026,321.596,-103.406,173.569,35.466,156.636
C09734=1060.032,321.843,-103.439,173.573,35.470,156.637
C09735=1060.039,322.091,-103.474,173.576,35.474,156.638
C09736=1060.045,322.339,-103.508,173.580,35.479,156.639
C09737=1060.052,322.586,-103.542,173.583,35.483,156.640
C09738=1060.058,322.834,-103.576,173.587,35.488,156.641
C09739=1060.065,323.081,-103.609,173.591,35.492,156.642
C09740=1060.071,323.329,-103.644,173.594,35.496,156.643
C09741=1060.079,323.577,-103.678,173.598,35.501,156.644
C09742=1060.085,323.824,-103.712,173.601,35.505,156.645
C09743=1060.091,324.072,-103.746,173.604,35.510,156.646
C09744=1060.098,324.319,-103.780,173.608,35.514,156.647
C09745=1060.104,324.567,-103.814,173.611,35.518,156.648
C09746=1060.111,324.815,-103.848,173.616,35.523,156.649
C09747=1060.117,325.062,-103.882,173.619,35.527,156.649
C09748=1060.124,325.310,-103.916,173.623,35.532,156.650
C09749=1060.131,325.557,-103.951,173.626,35.536,156.652
C09750=1060.138,325.805,-103.985,173.629,35.540,156.652
C09751=1060.143,326.052,-104.019,173.633,35.545,156.653
C09752=1060.151,326.300,-104.053,173.637,35.549,156.654
C09753=1060.157,326.548,-104.088,173.641,35.554,156.655
C09754=1060.164,326.796,-104.121,173.644,35.558,156.656
C09755=1060.170,327.042,-104.156,173.648,35.563,156.657
C09756=1060.177,327.290,-104.191,173.651,35.567,156.658
C09757=1060.184,327.538,-104.224,173.654,35.571,156.659
C09758=1060.191,327.786,-104.259,173.659,35.576,156.660
C09759=1060.197,328.033,-104.294,173.662,35.580,156.661
C09760=1060.204,328.280,-104.327,173.666,35.585,156.662
C09761=1060.210,328.528,-104.362,173.669,35.589,156.663
C09762=1060.217,328.776,-104.397,173.673,35.594,156.664
C09763=1060.224,329.023,-104.431,173.677,35.598,156.665
C09764=1060.231,329.271,-104.466,173.681,35.602,156.666
C09765=1060.237,329.518,-104.500,173.684,35.607,156.667
C09766=1060.244,329.766,-104.534,173.687,35.612,156.668
C09767=1060.251,330.013,-104.569,173.692,35.616,156.669
C09768=1060.257,330.261,-104.603,173.695,35.620,156.670
C09769=1060.265,330.508,-104.638,173.699,35.625,156.671
C09770=1060.271,330.756,-104.672,173.702,35.630,156.672
C09771=1060.278,331.004,-104.707,173.707,35.634,156.673
C09772=1060.284,331.251,-104.742,173.710,35.639,156.674
C09773=1060.291,331.496,-104.776,173.714,35.643,156.675
C09774=1060.297,331.741,-104.811,173.717,35.648,156.676
C09775=1060.304,331.986,-104.845,173.721,35.653,156.677
C09776=1060.310,332.230,-104.879,173.725,35.657,156.678
C09777=1060.317,332.474,-104.914,173.729,35.662,156.679
C09778=1060.323,332.719,-104.949,173.732,35.666,156.680
C09779=1060.330,332.964,-104.984,173.735,35.671,156.681
C09780=1060.336,333.210,-105.019,173.739,35.675,156.682
C09781=1060.342,333.456,-105.053,173.743,35.680,156.683
C09782=1060.349,333.704,-105.088,173.747,35.685,156.684
C09783=1060.355,333.952,-105.123,173.750,35.689,156.685
C09784=1060.362,334.199,-105.158,173.755,35.694,156.686
C09785=1060.369,334.446,-105.193,173.758,35.699,156.687
C09786=1060.376,334.694,-105.228,173.762,35.704,156.688
C09787=1060.382,334.942,-105.263,173.765,35.708,156.689
C09788=1060.389,335.189,-105.298,173.770,35.713,156.690
C09789=1060.396,335.437,-105.333,173.773,35.717,156.691
C09790=1060.402,335.684,-105.368,173.777,35.722,156.692
C09791=1060.409,335.931,-105.403,173.781,35.727,156.693
C09792=1060.416,336.179,-105.438,173.785,35.732,156.694
C09793=1060.422,336.426,-105.474,173.788,35.736,156.695
C09794=1060.429,336.674,-105.509,173.793,35.741,156.696
C09795=1060.435,336.921,-105.544,173.796,35.746,156.697
C09796=1060.442,337.168,-105.580,173.800,35.751,156.698
C09797=1060.449,337.416,-105.615,173.804,35.755,156.699
C09798=1060.455,337.663,-105.650,173.808,35.760,156.701
C09799=1060.462,337.911,-105.686,173.811,35.765,156.702
C09800=1060.469,338.158,-105.721,173.816,35.770,156.703
C09801=1060.475,338.406,-105.756,173.819,35.775,156.704
C09802=1060.482,338.653,-105.792,173.823,35.780,156.705
C09803=1060.489,338.901,-105.828,173.827,35.784,156.706
C09804=1060.495,339.148,-105.864,173.831,35.789,156.707
C09805=1060.502,339.396,-105.899,173.834,35.794,156.708
C09806=1060.509,339.643,-105.934,173.839,35.799,156.709
C09807=1060.515,339.890,-105.970,173.843,35.804,156.710
C09808=1060.522,340.138,-106.005,173.846,35.808,156.711
C09809=1060.528,340.385,-106.041,173.851,35.813,156.712
C09810=1060.535,340.633,-106.076,173.854,35.818,156.713
C09811=1060.542,340.879,-106.112,173.858,35.823,156.714
C09812=1060.549,341.127,-106.148,173.862,35.828,156.715
C09813=1060.555,341.375,-106.183,173.866,35.833,156.717
C09814=1060.562,341.622,-106.219,173.870,35.837,156.718
C09815=1060.569,341.869,-106.254,173.874,35.842,156.719
C09816=1060.575,342.116,-106.291,173.877,35.848,156.720
C09817=1060.583,342.364,-106.326,173.882,35.852,156.721
C09818=1060.590,342.611,-106.362,173.885,35.857,156.722
C09819=1060.596,342.859,-106.398,173.890,35.862,156.723
C09820=1060.603,343.105,-106.434,173.894,35.867,156.724
C09821=1060.609,343.354,-106.470,173.898,35.872,156.725
C09822=1060.616,343.601,-106.506,173.902,35.877,156.726
C09823=1060.622,343.848,-106.541,173.905,35.882,156.728
C09824=1060.630,344.095,-106.577,173.910,35.887,156.729
C09825=1060.636,344.343,-106.613,173.913,35.892,156.730
C09826=1060.643,344.590,-106.649,173.918,35.897,156.731
C09827=1060.650,344.837,-106.686,173.921,35.902,156.732
C09828=1060.656,345.085,-106.721,173.926,35.907,156.733
C09829=1060.663,345.351,-106.760,173.930,35.912,156.734
C09830=1060.671,345.616,-106.799,173.934,35.917,156.736
C09831=1060.678,345.883,-106.838,173.939,35.923,156.737
C09832=1060.685,346.149,-106.877,173.943,35.928,156.738
C09833=1060.692,346.395,-106.913,173.947,35.933,156.739
C09834=1060.698,346.643,-106.949,173.952,35.938,156.740
C09835=1060.705,346.891,-106.986,173.955,35.944,156.741
C09836=1060.712,347.138,-107.022,173.960,35.949,156.743
C09837=1060.718,347.385,-107.058,173.963,35.954,156.744
C09838=1060.725,347.632,-107.095,173.967,35.959,156.745
C09839=1060.732,347.879,-107.131,173.972,35.964,156.746
C09840=1060.739,348.126,-107.167,173.976,35.969,156.747
C09841=1060.746,348.374,-107.204,173.980,35.974,156.748
C09842=1060.753,348.621,-107.240,173.984,35.979,156.749
C09843=1060.760,348.869,-107.277,173.988,35.984,156.751
C09844=1060.766,349.116,-107.313,173.993,35.989,156.752
C09845=1060.772,349.363,-107.349,173.996,35.995,156.753
C09846=1060.780,349.610,-107.386,174.001,36.000,156.754
C09847=1060.786,349.857,-107.422,174.004,36.005,156.755
C09848=1060.793,350.105,-107.459,174.009,36.010,156.756
C09849=1060.800,350.352,-107.495,174.013,36.015,156.758
C09850=1060.807,350.599,-107.532,174.017,36.021,156.759
C09851=1060.814,350.846,-107.568,174.021,36.026,156.760
C09852=1060.821,351.094,-107.605,174.025,36.031,156.761
C09853=1060.827,351.341,-107.642,174.030,36.036,156.762
C09854=1060.835,351.588,-107.678,174.034,36.041,156.764
C09855=1060.841,351.835,-107.715,174.038,36.047,156.765
C09856=1060.848,352.083,-107.751,174.042,36.052,156.766
C09857=1060.855,352.329,-107.789,174.047,36.057,156.767
C09858=1060.862,352.577,-107.825,174.050,36.062,156.768
C09859=1060.868,352.824,-107.862,174.055,36.068,156.770
C09860=1060.875,353.071,-107.899,174.059,36.073,156.771
C09861=1060.881,353.305,-107.934,174.063,36.078,156.772
C09862=1060.888,353.538,-107.969,174.067,36.083,156.773
C09863=1060.894,353.770,-108.004,174.071,36.088,156.774
C09864=1060.901,354.004,-108.038,174.075,36.093,156.775
C09865=1060.907,354.236,-108.073,174.080,36.098,156.776
C09866=1060.914,354.469,-108.108,174.083,36.104,156.778
C09867=1060.920,354.703,-108.143,174.087,36.109,156.779
C09868=1060.927,354.936,-108.178,174.091,36.114,156.780
C09869=1060.933,355.182,-108.215,174.095,36.119,156.781
C09870=1060.940,355.430,-108.252,174.100,36.124,156.782
C09871=1060.947,355.677,-108.289,174.104,36.129,156.784
C09872=1060.953,355.924,-108.326,174.108,36.135,156.785
C09873=1060.961,356.172,-108.364,174.113,36.141,156.786
C09874=1060.967,356.418,-108.401,174.117,36.146,156.787
C09875=1060.974,356.666,-108.438,174.121,36.151,156.789
C09876=1060.982,356.913,-108.475,174.126,36.156,156.790
C09877=1060.988,357.159,-108.512,174.130,36.162,156.791
C09878=1060.995,357.406,-108.550,174.134,36.168,156.792
C09879=1061.002,357.654,-108.587,174.139,36.173,156.794
C09880=1061.010,357.901,-108.624,174.143,36.178,156.795
C09881=1061.016,358.148,-108.661,174.147,36.184,156.796
C09882=1061.023,358.395,-108.699,174.152,36.190,156.797
C09883=1061.031,358.642,-108.736,174.157,36.195,156.799
C09884=1061.037,358.889,-108.773,174.160,36.201,156.800
C09885=1061.044,359.134,-108.811,174.165,36.206,156.801
C09886=1061.051,359.378,-108.848,174.170,36.211,156.802
C09887=1061.058,359.623,-108.885,174.173,36.217,156.804
C09888=1061.064,359.868,-108.922,174.178,36.223,156.805
C09889=1061.071,360.113,-108.959,174.183,36.228,156.806
C09890=1061.079,360.357,-108.997,174.188,36.234,156.808
C09891=1061.086,360.602,-109.034,174.191,36.239,156.809
C09892=1061.092,360.846,-109.071,174.196,36.244,156.810
C09893=1061.099,361.093,-109.109,174.201,36.250,156.811
C09894=1061.106,361.340,-109.146,174.204,36.256,156.813
C09895=1061.113,361.588,-109.184,174.209,36.262,156.814
C09896=1061.120,361.834,-109.222,174.214,36.267,156.815
C09897=1061.127,362.082,-109.260,174.219,36.273,156.817
C09898=1061.135,362.329,-109.297,174.222,36.279,156.818
C09899=1061.141,362.575,-109.335,174.227,36.284,156.819
C09900=1061.148,362.823,-109.373,174.232,36.290,156.821
C09901=1061.155,363.069,-109.411,174.236,36.295,156.822
C09902=1061.162,363.317,-109.449,174.241,36.301,156.823
C09903=1061.169,363.564,-109.487,174.245,36.307,156.825
C09904=1061.177,363.810,-109.525,174.250,36.313,156.826
C09905=1061.183,364.058,-109.563,174.255,36.318,156.827
C09906=1061.190,364.305,-109.601,174.259,36.324,156.829
C09907=1061.197,364.552,-109.639,174.264,36.330,156.830
C09908=1061.204,364.799,-109.677,174.268,36.336,156.831
C09909=1061.211,365.045,-109.715,174.273,36.342,156.833
C09910=1061.218,365.292,-109.753,174.277,36.348,156.834
C09911=1061.225,365.539,-109.792,174.282,36.353,156.835
C09912=1061.231,365.786,-109.830,174.287,36.359,156.837
C09913=1061.239,366.033,-109.868,174.291,36.365,156.838
C09914=1061.245,366.280,-109.906,174.296,36.371,156.840
C09915=1061.253,366.527,-109.944,174.300,36.377,156.841
C09916=1061.260,366.774,-109.983,174.305,36.383,156.842
C09917=1061.267,367.021,-110.021,174.310,36.389,156.844
C09918=1061.274,367.268,-110.060,174.315,36.395,156.845
C09919=1061.280,367.514,-110.099,174.320,36.401,156.846
C09920=1061.288,367.761,-110.136,174.323,36.407,156.848
C09921=1061.295,368.008,-110.175,174.328,36.412,156.849
C09922=1061.302,368.255,-110.213,174.333,36.418,156.851
C09923=1061.309,368.502,-110.252,174.338,36.425,156.852
C09924=1061.316,368.750,-110.290,174.343,36.431,156.853
C09925=1061.324,368.996,-110.329,174.347,36.436,156.855
C09926=1061.330,369.243,-110.368,174.352,36.442,156.856
C09927=1061.338,369.490,-110.406,174.357,36.448,156.858
C09928=1061.345,369.736,-110.445,174.362,36.455,156.859
C09929=1061.352,369.983,-110.483,174.367,36.461,156.861
C09930=1061.359,370.230,-110.522,174.371,36.467,156.862
C09931=1061.367,370.477,-110.561,174.375,36.472,156.863
C09932=1061.373,370.724,-110.600,174.380,36.478,156.865
C09933=1061.381,370.971,-110.638,174.385,36.485,156.866
C09934=1061.388,371.218,-110.677,174.390,36.491,156.868
C09935=1061.394,371.464,-110.716,174.395,36.497,156.869
C09936=1061.403,371.712,-110.754,174.400,36.503,156.870
C09937=1061.409,371.958,-110.793,174.405,36.509,156.872
C09938=1061.416,372.205,-110.832,174.409,36.515,156.873
C09939=1061.424,372.452,-110.871,174.414,36.522,156.875
C09940=1061.431,372.699,-110.909,174.419,36.528,156.876
C09941=1061.439,372.959,-110.951,174.424,36.534,156.878
C09942=1061.446,373.220,-110.992,174.429,36.541,156.880
C09943=1061.454,373.480,-111.034,174.435,36.548,156.881
C09944=1061.461,373.741,-111.075,174.440,36.554,156.883
C09945=1061.468,373.988,-111.114,174.445,36.560,156.884
C09946=1061.475,374.234,-111.153,174.450,36.566,156.886
C09947=1061.482,374.481,-111.192,174.455,36.573,156.887
C09948=1061.490,374.728,-111.232,174.460,36.579,156.889
C09949=1061.497,374.974,-111.271,174.465,36.586,156.890
C09950=1061.504,375.221,-111.310,174.469,36.592,156.892
C09951=1061.511,375.468,-111.350,174.474,36.598,156.893
C09952=1061.518,375.714,-111.389,174.479,36.604,156.895
C09953=1061.525,375.961,-111.428,174.484,36.611,156.896
C09954=1061.533,376.208,-111.468,174.489,36.617,156.898
C09955=1061.540,376.455,-111.507,174.494,36.624,156.899
C09956=1061.547,376.701,-111.546,174.499,36.630,156.901
C09957=1061.554,376.948,-111.586,174.504,36.636,156.902
C09958=1061.561,377.195,-111.625,174.509,36.643,156.904
C09959=1061.569,377.442,-111.665,174.514,36.650,156.905
C09960=1061.576,377.688,-111.704,174.520,36.656,156.907
C09961=1061.583,377.935,-111.744,174.525,36.662,156.908
C09962=1061.591,378.182,-111.783,174.530,36.669,156.910
C09963=1061.598,378.429,-111.823,174.535,36.676,156.912
C09964=1061.605,378.675,-111.863,174.540,36.682,156.913
C09965=1061.613,378.922,-111.903,174.545,36.689,156.915
C09966=1061.620,379.168,-111.941,174.550,36.695,156.916
C09967=1061.628,379.415,-111.981,174.555,36.701,156.918
C09968=1061.635,379.662,-112.021,174.560,36.708,156.919
C09969=1061.643,379.908,-112.061,174.566,36.715,156.921
C09970=1061.650,380.155,-112.100,174.571,36.721,156.923
C09971=1061.657,380.402,-112.140,174.576,36.728,156.924
C09972=1061.665,380.649,-112.180,174.581,36.734,156.926
C09973=1061.672,380.895,-112.220,174.586,36.741,156.928
C09974=1061.679,381.142,-112.260,174.591,36.748,156.929
C09975=1061.686,381.388,-112.300,174.597,36.755,156.931
C09976=1061.694,381.635,-112.340,174.602,36.761,156.932
C09977=1061.701,381.881,-112.381,174.607,36.768,156.934
C09978=1061.708,382.128,-112.421,174.612,36.775,156.936
C09979=1061.716,382.375,-112.460,174.617,36.781,156.937
C09980=1061.723,382.621,-112.501,174.623,36.789,156.939
C09981=1061.731,382.868,-112.541,174.628,36.795,156.941
C09982=1061.737,383.114,-112.581,174.633,36.802,156.942
C09983=1061.745,383.361,-112.621,174.638,36.809,156.944
C09984=1061.753,383.607,-112.662,174.643,36.816,156.946
C09985=1061.759,383.854,-112.702,174.649,36.822,156.947
C09986=1061.767,384.100,-112.743,174.654,36.830,156.949
C09987=1061.775,384.347,-112.783,174.659,36.837,156.951
C09988=1061.782,384.594,-112.823,174.664,36.843,156.952
C09989=1061.789,384.840,-112.863,174.670,36.850,156.954
C09990=1061.796,385.087,-112.904,174.676,36.857,156.956
C09991=1061.804,385.333,-112.945,174.681,36.864,156.957
C09992=1061.812,385.580,-112.985,174.686,36.871,156.959
C09993=1061.819,385.826,-113.025,174.692,36.878,156.961
C09994=1061.827,386.072,-113.066,174.697,36.885,156.962
C09995=1061.834,386.320,-113.106,174.702,36.892,156.964
C09996=1061.842,386.566,-113.147,174.708,36.899,156.966
//INST
///DATE 2021/06/17 10:56
///ATTR SC,RW,RJ
////FRAME ROBOT
///GROUP1 RB1
NOP
MOVL C00000 V=800.0 PL=0
MOVL C00001 V=800.0 PL=0
MOVL C00002 V=800.0 PL=0
MOVL C00003 V=800.0 PL=0
MOVL C00004 V=800.0 PL=0
MOVL C00005 V=800.0 PL=0
MOVL C00006 V=800.0 PL=0
MOVL C00007 V=800.0 PL=0
MOVL C00008 V=800.0 PL=0
MOVL C00009 V=800.0 PL=0
MOVL C00010 V=800.0 PL=0
MOVL C00011 V=800.0 PL=0
MOVL C00012 V=800.0 PL=0
MOVL C00013 V=800.0 PL=0
MOVL C00014 V=800.0 PL=0
MOVL C00015 V=800.0 PL=0
MOVL C00016 V=800.0 PL=0
MOVL C00017 V=800.0 PL=0
MOVL C00018 V=800.0 PL=0
MOVL C00019 V=800.0 PL=0
MOVL C00020 V=800.0 PL=0
MOVL C00021 V=800.0 PL=0
MOVL C00022 V=800.0 PL=0
MOVL C00023 V=800.0 PL=0
MOVL C00024 V=800.0 PL=0
MOVL C00025 V=800.0 PL=0
MOVL C00026 V=800.0 PL=0
MOVL C00027 V=800.0 PL=0
MOVL C00028 V=800.0 PL=0
MOVL C00029 V=800.0 PL=0
MOVL C00030 V=800.0 PL=0
MOVL C00031 V=800.0 PL=0
MOVL C00032 V=800.0 PL=0
MOVL C00033 V=800.0 PL=0
MOVL C00034 V=800.0 PL=0
MOVL C00035 V=800.0 PL=0
MOVL C00036 V=800.0 PL=0
MOVL C00037 V=800.0 PL=0
MOVL C00038 V=800.0 PL=0
MOVL C00039 V=800.0 PL=0
MOVL C00040 V=800.0 PL=0
MOVL C00041 V=800.0 PL=0
MOVL C00042 V=800.0 PL=0
MOVL C00043 V=800.0 PL=0
MOVL C00044 V=800.0 PL=0
MOVL C00045 V=800.0 PL=0
MOVL C00046 V=800.0 PL=0
MOVL C00047 V=800.0 PL=0
MOVL C00048 V=800.0 PL=0
MOVL C00049 V=800.0 PL=0
MOVL C00050 V=800.0 PL=0
MOVL C00051 V=800.0 PL=0
MOVL C00052 V=800.0 PL=0
MOVL C00053 V=800.0 PL=0
MOVL C00054 V=800.0 PL=0
MOVL C00055 V=800.0 PL=0
MOVL C00056 V=800.0 PL=0
MOVL C00057 V=800.0 PL=0
MOVL C00058 V=800.0 PL=0
MOVL C00059 V=800.0 PL=0
MOVL C00060 V=800.0 PL=0
MOVL C00061 V=800.0 PL=0
MOVL C00062 V=800.0 PL=0
MOVL C00063 V=800.0 PL=0
MOVL C00064 V=800.0 PL=0
MOVL C00065 V=800.0 PL=0
MOVL C00066 V=800.0 PL=0
MOVL C00067 V=800.0 PL=0
MOVL C00068 V=800.0 PL=0
MOVL C00069 V=800.0 PL=0
MOVL C00070 V=800.0 PL=0
MOVL C00071 V=800.0 PL=0
MOVL C00072 V=800.0 PL=0
MOVL C00073 V=800.0 PL=0
MOVL C00074 V=800.0 PL=0
MOVL C00075 V=800.0 PL=0
MOVL C00076 V=800.0 PL=0
MOVL C00077 V=800.0 PL=0
MOVL C00078 V=800.0 PL=0
MOVL C00079 V=800.0 PL=0
MOVL C00080 V=800.0 PL=0
MOVL C00081 V=800.0 PL=0
MOVL C00082 V=800.0 PL=0
MOVL C00083 V=800.0 PL=0
MOVL C00084 V=800.0 PL=0
MOVL C00085 V=800.0 PL=0
MOVL C00086 V=800.0 PL=0
MOVL C00087 V=800.0 PL=0
MOVL C00088 V=800.0 PL=0
MOVL C00089 V=800.0 PL=0
MOVL C00090 V=800.0 PL=0
MOVL C00091 V=800.0 PL=0
MOVL C00092 V=800.0 PL=0
MOVL C00093 V=800.0 PL=0
MOVL C00094 V=800.0 PL=0
MOVL C00095 V=800.0 PL=0
MOVL C00096 V=800.0 PL=0
MOVL C00097 V=800.0 PL=0
MOVL C00098 V=800.0 PL=0
MOVL C00099 V=800.0 PL=0
MOVL C00100 V=800.0 PL=0
MOVL C00101 V=800.0 PL=0
MOVL C00102 V=800.0 PL=0
MOVL C00103 V=800.0 PL=0
MOVL C00104 V=800.0 PL=0
MOVL C00105 V=800.0 PL=0
MOVL C00106 V=800.0 PL=0
MOVL C00107 V=800.0 PL=0
MOVL C00108 V=800.0 PL=0
MOVL C00109 V=800.0 PL=0
MOVL C00110 V=800.0 PL=0
MOVL C00111 V=800.0 PL=0
MOVL C00112 V=800.0 PL=0
MOVL C00113 V=800.0 PL=0
MOVL C00114 V=800.0 PL=0
MOVL C00115 V=800.0 PL=0
MOVL C00116 V=800.0 PL=0
MOVL C00117 V=800.0 PL=0
MOVL C00118 V=800.0 PL=0
MOVL C00119 V=800.0 PL=0
MOVL C00120 V=800.0 PL=0
MOVL C00121 V=800.0 PL=0
MOVL C00122 V=800.0 PL=0
MOVL C00123 V=800.0 PL=0
MOVL C00124 V=800.0 PL=0
MOVL C00125 V=800.0 PL=0
MOVL C00126 V=800.0 PL=0
MOVL C00127 V=800.0 PL=0
MOVL C00128 V=800.0 PL=0
MOVL C00129 V=800.0 PL=0
MOVL C00130 V=800.0 PL=0
MOVL C00131 V=800.0 PL=0
MOVL C00132 V=800.0 PL=0
MOVL C00133 V=800.0 PL=0
MOVL C00134 V=800.0 PL=0
MOVL C00135 V=800.0 PL=0
MOVL C00136 V=800.0 PL=0
MOVL C00137 V=800.0 PL=0
MOVL C00138 V=800.0 PL=0
MOVL C00139 V=800.0 PL=0
MOVL C00140 V=800.0 PL=0
MOVL C00141 V=800.0 PL=0
MOVL C00142 V=800.0 PL=0
MOVL C00143 V=800.0 PL=0
MOVL C00144 V=800.0 PL=0
MOVL C00145 V=800.0 PL=0
MOVL C00146 V=800.0 PL=0
MOVL C00147 V=800.0 PL=0
MOVL C00148 V=800.0 PL=0
MOVL C00149 V=800.0 PL=0
MOVL C00150 V=800.0 PL=0
MOVL C00151 V=800.0 PL=0
MOVL C00152 V=800.0 PL=0
MOVL C00153 V=800.0 PL=0
MOVL C00154 V=800.0 PL=0
MOVL C00155 V=800.0 PL=0
MOVL C00156 V=800.0 PL=0
MOVL C00157 V=800.0 PL=0
MOVL C00158 V=800.0 PL=0
MOVL C00159 V=800.0 PL=0
MOVL C00160 V=800.0 PL=0
MOVL C00161 V=800.0 PL=0
MOVL C00162 V=800.0 PL=0
MOVL C00163 V=800.0 PL=0
MOVL C00164 V=800.0 PL=0
MOVL C00165 V=800.0 PL=0
MOVL C00166 V=800.0 PL=0
MOVL C00167 V=800.0 PL=0
MOVL C00168 V=800.0 PL=0
MOVL C00169 V=800.0 PL=0
MOVL C00170 V=800.0 PL=0
MOVL C00171 V=800.0 PL=0
MOVL C00172 V=800.0 PL=0
MOVL C00173 V=800.0 PL=0
MOVL C00174 V=800.0 PL=0
MOVL C00175 V=800.0 PL=0
MOVL C00176 V=800.0 PL=0
MOVL C00177 V=800.0 PL=0
MOVL C00178 V=800.0 PL=0
MOVL C00179 V=800.0 PL=0
MOVL C00180 V=800.0 PL=0
MOVL C00181 V=800.0 PL=0
MOVL C00182 V=800.0 PL=0
MOVL C00183 V=800.0 PL=0
MOVL C00184 V=800.0 PL=0
MOVL C00185 V=800.0 PL=0
MOVL C00186 V=800.0 PL=0
MOVL C00187 V=800.0 PL=0
MOVL C00188 V=800.0 PL=0
MOVL C00189 V=800.0 PL=0
MOVL C00190 V=800.0 PL=0
MOVL C00191 V=800.0 PL=0
MOVL C00192 V=800.0 PL=0
MOVL C00193 V=800.0 PL=0
MOVL C00194 V=800.0 PL=0
MOVL C00195 V=800.0 PL=0
MOVL C00196 V=800.0 PL=0
MOVL C00197 V=800.0 PL=0
MOVL C00198 V=800.0 PL=0
MOVL C00199 V=800.0 PL=0
MOVL C00200 V=800.0 PL=0
MOVL C00201 V=800.0 PL=0
MOVL C00202 V=800.0 PL=0
MOVL C00203 V=800.0 PL=0
MOVL C00204 V=800.0 PL=0
MOVL C00205 V=800.0 PL=0
MOVL C00206 V=800.0 PL=0
MOVL C00207 V=800.0 PL=0
MOVL C00208 V=800.0 PL=0
MOVL C00209 V=800.0 PL=0
MOVL C00210 V=800.0 PL=0
MOVL C00211 V=800.0 PL=0
MOVL C00212 V=800.0 PL=0
MOVL C00213 V=800.0 PL=0
MOVL C00214 V=800.0 PL=0
MOVL C00215 V=800.0 PL=0
MOVL C00216 V=800.0 PL=0
MOVL C00217 V=800.0 PL=0
MOVL C00218 V=800.0 PL=0
MOVL C00219 V=800.0 PL=0
MOVL C00220 V=800.0 PL=0
MOVL C00221 V=800.0 PL=0
MOVL C00222 V=800.0 PL=0
MOVL C00223 V=800.0 PL=0
MOVL C00224 V=800.0 PL=0
MOVL C00225 V=800.0 PL=0
MOVL C00226 V=800.0 PL=0
MOVL C00227 V=800.0 PL=0
MOVL C00228 V=800.0 PL=0
MOVL C00229 V=800.0 PL=0
MOVL C00230 V=800.0 PL=0
MOVL C00231 V=800.0 PL=0
MOVL C00232 V=800.0 PL=0
MOVL C00233 V=800.0 PL=0
MOVL C00234 V=800.0 PL=0
MOVL C00235 V=800.0 PL=0
MOVL C00236 V=800.0 PL=0
MOVL C00237 V=800.0 PL=0
MOVL C00238 V=800.0 PL=0
MOVL C00239 V=800.0 PL=0
MOVL C00240 V=800.0 PL=0
MOVL C00241 V=800.0 PL=0
MOVL C00242 V=800.0 PL=0
MOVL C00243 V=800.0 PL=0
MOVL C00244 V=800.0 PL=0
MOVL C00245 V=800.0 PL=0
MOVL C00246 V=800.0 PL=0
MOVL C00247 V=800.0 PL=0
MOVL C00248 V=800.0 PL=0
MOVL C00249 V=800.0 PL=0
MOVL C00250 V=800.0 PL=0
MOVL C00251 V=800.0 PL=0
MOVL C00252 V=800.0 PL=0
MOVL C00253 V=800.0 PL=0
MOVL C00254 V=800.0 PL=0
MOVL C00255 V=800.0 PL=0
MOVL C00256 V=800.0 PL=0
MOVL C00257 V=800.0 PL=0
MOVL C00258 V=800.0 PL=0
MOVL C00259 V=800.0 PL=0
MOVL C00260 V=800.0 PL=0
MOVL C00261 V=800.0 PL=0
MOVL C00262 V=800.0 PL=0
MOVL C00263 V=800.0 PL=0
MOVL C00264 V=800.0 PL=0
MOVL C00265 V=800.0 PL=0
MOVL C00266 V=800.0 PL=0
MOVL C00267 V=800.0 PL=0
MOVL C00268 V=800.0 PL=0
MOVL C00269 V=800.0 PL=0
MOVL C00270 V=800.0 PL=0
MOVL C00271 V=800.0 PL=0
MOVL C00272 V=800.0 PL=0
MOVL C00273 V=800.0 PL=0
MOVL C00274 V=800.0 PL=0
MOVL C00275 V=800.0 PL=0
MOVL C00276 V=800.0 PL=0
MOVL C00277 V=800.0 PL=0
MOVL C00278 V=800.0 PL=0
MOVL C00279 V=800.0 PL=0
MOVL C00280 V=800.0 PL=0
MOVL C00281 V=800.0 PL=0
MOVL C00282 V=800.0 PL=0
MOVL C00283 V=800.0 PL=0
MOVL C00284 V=800.0 PL=0
MOVL C00285 V=800.0 PL=0
MOVL C00286 V=800.0 PL=0
MOVL C00287 V=800.0 PL=0
MOVL C00288 V=800.0 PL=0
MOVL C00289 V=800.0 PL=0
MOVL C00290 V=800.0 PL=0
MOVL C00291 V=800.0 PL=0
MOVL C00292 V=800.0 PL=0
MOVL C00293 V=800.0 PL=0
MOVL C00294 V=800.0 PL=0
MOVL C00295 V=800.0 PL=0
MOVL C00296 V=800.0 PL=0
MOVL C00297 V=800.0 PL=0
MOVL C00298 V=800.0 PL=0
MOVL C00299 V=800.0 PL=0
MOVL C00300 V=800.0 PL=0
MOVL C00301 V=800.0 PL=0
MOVL C00302 V=800.0 PL=0
MOVL C00303 V=800.0 PL=0
MOVL C00304 V=800.0 PL=0
MOVL C00305 V=800.0 PL=0
MOVL C00306 V=800.0 PL=0
MOVL C00307 V=800.0 PL=0
MOVL C00308 V=800.0 PL=0
MOVL C00309 V=800.0 PL=0
MOVL C00310 V=800.0 PL=0
MOVL C00311 V=800.0 PL=0
MOVL C00312 V=800.0 PL=0
MOVL C00313 V=800.0 PL=0
MOVL C00314 V=800.0 PL=0
MOVL C00315 V=800.0 PL=0
MOVL C00316 V=800.0 PL=0
MOVL C00317 V=800.0 PL=0
MOVL C00318 V=800.0 PL=0
MOVL C00319 V=800.0 PL=0
MOVL C00320 V=800.0 PL=0
MOVL C00321 V=800.0 PL=0
MOVL C00322 V=800.0 PL=0
MOVL C00323 V=800.0 PL=0
MOVL C00324 V=800.0 PL=0
MOVL C00325 V=800.0 PL=0
MOVL C00326 V=800.0 PL=0
MOVL C00327 V=800.0 PL=0
MOVL C00328 V=800.0 PL=0
MOVL C00329 V=800.0 PL=0
MOVL C00330 V=800.0 PL=0
MOVL C00331 V=800.0 PL=0
MOVL C00332 V=800.0 PL=0
MOVL C00333 V=800.0 PL=0
MOVL C00334 V=800.0 PL=0
MOVL C00335 V=800.0 PL=0
MOVL C00336 V=800.0 PL=0
MOVL C00337 V=800.0 PL=0
MOVL C00338 V=800.0 PL=0
MOVL C00339 V=800.0 PL=0
MOVL C00340 V=800.0 PL=0
MOVL C00341 V=800.0 PL=0
MOVL C00342 V=800.0 PL=0
MOVL C00343 V=800.0 PL=0
MOVL C00344 V=800.0 PL=0
MOVL C00345 V=800.0 PL=0
MOVL C00346 V=800.0 PL=0
MOVL C00347 V=800.0 PL=0
MOVL C00348 V=800.0 PL=0
MOVL C00349 V=800.0 PL=0
MOVL C00350 V=800.0 PL=0
MOVL C00351 V=800.0 PL=0
MOVL C00352 V=800.0 PL=0
MOVL C00353 V=800.0 PL=0
MOVL C00354 V=800.0 PL=0
MOVL C00355 V=800.0 PL=0
MOVL C00356 V=800.0 PL=0
MOVL C00357 V=800.0 PL=0
MOVL C00358 V=800.0 PL=0
MOVL C00359 V=800.0 PL=0
MOVL C00360 V=800.0 PL=0
MOVL C00361 V=800.0 PL=0
MOVL C00362 V=800.0 PL=0
MOVL C00363 V=800.0 PL=0
MOVL C00364 V=800.0 PL=0
MOVL C00365 V=800.0 PL=0
MOVL C00366 V=800.0 PL=0
MOVL C00367 V=800.0 PL=0
MOVL C00368 V=800.0 PL=0
MOVL C00369 V=800.0 PL=0
MOVL C00370 V=800.0 PL=0
MOVL C00371 V=800.0 PL=0
MOVL C00372 V=800.0 PL=0
MOVL C00373 V=800.0 PL=0
MOVL C00374 V=800.0 PL=0
MOVL C00375 V=800.0 PL=0
MOVL C00376 V=800.0 PL=0
MOVL C00377 V=800.0 PL=0
MOVL C00378 V=800.0 PL=0
MOVL C00379 V=800.0 PL=0
MOVL C00380 V=800.0 PL=0
MOVL C00381 V=800.0 PL=0
MOVL C00382 V=800.0 PL=0
MOVL C00383 V=800.0 PL=0
MOVL C00384 V=800.0 PL=0
MOVL C00385 V=800.0 PL=0
MOVL C00386 V=800.0 PL=0
MOVL C00387 V=800.0 PL=0
MOVL C00388 V=800.0 PL=0
MOVL C00389 V=800.0 PL=0
MOVL C00390 V=800.0 PL=0
MOVL C00391 V=800.0 PL=0
MOVL C00392 V=800.0 PL=0
MOVL C00393 V=800.0 PL=0
MOVL C00394 V=800.0 PL=0
MOVL C00395 V=800.0 PL=0
MOVL C00396 V=800.0 PL=0
MOVL C00397 V=800.0 PL=0
MOVL C00398 V=800.0 PL=0
MOVL C00399 V=800.0 PL=0
MOVL C00400 V=800.0 PL=0
MOVL C00401 V=800.0 PL=0
MOVL C00402 V=800.0 PL=0
MOVL C00403 V=800.0 PL=0
MOVL C00404 V=800.0 PL=0
MOVL C00405 V=800.0 PL=0
MOVL C00406 V=800.0 PL=0
MOVL C00407 V=800.0 PL=0
MOVL C00408 V=800.0 PL=0
MOVL C00409 V=800.0 PL=0
MOVL C00410 V=800.0 PL=0
MOVL C00411 V=800.0 PL=0
MOVL C00412 V=800.0 PL=0
MOVL C00413 V=800.0 PL=0
MOVL C00414 V=800.0 PL=0
MOVL C00415 V=800.0 PL=0
MOVL C00416 V=800.0 PL=0
MOVL C00417 V=800.0 PL=0
MOVL C00418 V=800.0 PL=0
MOVL C00419 V=800.0 PL=0
MOVL C00420 V=800.0 PL=0
MOVL C00421 V=800.0 PL=0
MOVL C00422 V=800.0 PL=0
MOVL C00423 V=800.0 PL=0
MOVL C00424 V=800.0 PL=0
MOVL C00425 V=800.0 PL=0
MOVL C00426 V=800.0 PL=0
MOVL C00427 V=800.0 PL=0
MOVL C00428 V=800.0 PL=0
MOVL C00429 V=800.0 PL=0
MOVL C00430 V=800.0 PL=0
MOVL C00431 V=800.0 PL=0
MOVL C00432 V=800.0 PL=0
MOVL C00433 V=800.0 PL=0
MOVL C00434 V=800.0 PL=0
MOVL C00435 V=800.0 PL=0
MOVL C00436 V=800.0 PL=0
MOVL C00437 V=800.0 PL=0
MOVL C00438 V=800.0 PL=0
MOVL C00439 V=800.0 PL=0
MOVL C00440 V=800.0 PL=0
MOVL C00441 V=800.0 PL=0
MOVL C00442 V=800.0 PL=0
MOVL C00443 V=800.0 PL=0
MOVL C00444 V=800.0 PL=0
MOVL C00445 V=800.0 PL=0
MOVL C00446 V=800.0 PL=0
MOVL C00447 V=800.0 PL=0
MOVL C00448 V=800.0 PL=0
MOVL C00449 V=800.0 PL=0
MOVL C00450 V=800.0 PL=0
MOVL C00451 V=800.0 PL=0
MOVL C00452 V=800.0 PL=0
MOVL C00453 V=800.0 PL=0
MOVL C00454 V=800.0 PL=0
MOVL C00455 V=800.0 PL=0
MOVL C00456 V=800.0 PL=0
MOVL C00457 V=800.0 PL=0
MOVL C00458 V=800.0 PL=0
MOVL C00459 V=800.0 PL=0
MOVL C00460 V=800.0 PL=0
MOVL C00461 V=800.0 PL=0
MOVL C00462 V=800.0 PL=0
MOVL C00463 V=800.0 PL=0
MOVL C00464 V=800.0 PL=0
MOVL C00465 V=800.0 PL=0
MOVL C00466 V=800.0 PL=0
MOVL C00467 V=800.0 PL=0
MOVL C00468 V=800.0 PL=0
MOVL C00469 V=800.0 PL=0
MOVL C00470 V=800.0 PL=0
MOVL C00471 V=800.0 PL=0
MOVL C00472 V=800.0 PL=0
MOVL C00473 V=800.0 PL=0
MOVL C00474 V=800.0 PL=0
MOVL C00475 V=800.0 PL=0
MOVL C00476 V=800.0 PL=0
MOVL C00477 V=800.0 PL=0
MOVL C00478 V=800.0 PL=0
MOVL C00479 V=800.0 PL=0
MOVL C00480 V=800.0 PL=0
MOVL C00481 V=800.0 PL=0
MOVL C00482 V=800.0 PL=0
MOVL C00483 V=800.0 PL=0
MOVL C00484 V=800.0 PL=0
MOVL C00485 V=800.0 PL=0
MOVL C00486 V=800.0 PL=0
MOVL C00487 V=800.0 PL=0
MOVL C00488 V=800.0 PL=0
MOVL C00489 V=800.0 PL=0
MOVL C00490 V=800.0 PL=0
MOVL C00491 V=800.0 PL=0
MOVL C00492 V=800.0 PL=0
MOVL C00493 V=800.0 PL=0
MOVL C00494 V=800.0 PL=0
MOVL C00495 V=800.0 PL=0
MOVL C00496 V=800.0 PL=0
MOVL C00497 V=800.0 PL=0
MOVL C00498 V=800.0 PL=0
MOVL C00499 V=800.0 PL=0
MOVL C00500 V=800.0 PL=0
MOVL C00501 V=800.0 PL=0
MOVL C00502 V=800.0 PL=0
MOVL C00503 V=800.0 PL=0
MOVL C00504 V=800.0 PL=0
MOVL C00505 V=800.0 PL=0
MOVL C00506 V=800.0 PL=0
MOVL C00507 V=800.0 PL=0
MOVL C00508 V=800.0 PL=0
MOVL C00509 V=800.0 PL=0
MOVL C00510 V=800.0 PL=0
MOVL C00511 V=800.0 PL=0
MOVL C00512 V=800.0 PL=0
MOVL C00513 V=800.0 PL=0
MOVL C00514 V=800.0 PL=0
MOVL C00515 V=800.0 PL=0
MOVL C00516 V=800.0 PL=0
MOVL C00517 V=800.0 PL=0
MOVL C00518 V=800.0 PL=0
MOVL C00519 V=800.0 PL=0
MOVL C00520 V=800.0 PL=0
MOVL C00521 V=800.0 PL=0
MOVL C00522 V=800.0 PL=0
MOVL C00523 V=800.0 PL=0
MOVL C00524 V=800.0 PL=0
MOVL C00525 V=800.0 PL=0
MOVL C00526 V=800.0 PL=0
MOVL C00527 V=800.0 PL=0
MOVL C00528 V=800.0 PL=0
MOVL C00529 V=800.0 PL=0
MOVL C00530 V=800.0 PL=0
MOVL C00531 V=800.0 PL=0
MOVL C00532 V=800.0 PL=0
MOVL C00533 V=800.0 PL=0
MOVL C00534 V=800.0 PL=0
MOVL C00535 V=800.0 PL=0
MOVL C00536 V=800.0 PL=0
MOVL C00537 V=800.0 PL=0
MOVL C00538 V=800.0 PL=0
MOVL C00539 V=800.0 PL=0
MOVL C00540 V=800.0 PL=0
MOVL C00541 V=800.0 PL=0
MOVL C00542 V=800.0 PL=0
MOVL C00543 V=800.0 PL=0
MOVL C00544 V=800.0 PL=0
MOVL C00545 V=800.0 PL=0
MOVL C00546 V=800.0 PL=0
MOVL C00547 V=800.0 PL=0
MOVL C00548 V=800.0 PL=0
MOVL C00549 V=800.0 PL=0
MOVL C00550 V=800.0 PL=0
MOVL C00551 V=800.0 PL=0
MOVL C00552 V=800.0 PL=0
MOVL C00553 V=800.0 PL=0
MOVL C00554 V=800.0 PL=0
MOVL C00555 V=800.0 PL=0
MOVL C00556 V=800.0 PL=0
MOVL C00557 V=800.0 PL=0
MOVL C00558 V=800.0 PL=0
MOVL C00559 V=800.0 PL=0
MOVL C00560 V=800.0 PL=0
MOVL C00561 V=800.0 PL=0
MOVL C00562 V=800.0 PL=0
MOVL C00563 V=800.0 PL=0
MOVL C00564 V=800.0 PL=0
MOVL C00565 V=800.0 PL=0
MOVL C00566 V=800.0 PL=0
MOVL C00567 V=800.0 PL=0
MOVL C00568 V=800.0 PL=0
MOVL C00569 V=800.0 PL=0
MOVL C00570 V=800.0 PL=0
MOVL C00571 V=800.0 PL=0
MOVL C00572 V=800.0 PL=0
MOVL C00573 V=800.0 PL=0
MOVL C00574 V=800.0 PL=0
MOVL C00575 V=800.0 PL=0
MOVL C00576 V=800.0 PL=0
MOVL C00577 V=800.0 PL=0
MOVL C00578 V=800.0 PL=0
MOVL C00579 V=800.0 PL=0
MOVL C00580 V=800.0 PL=0
MOVL C00581 V=800.0 PL=0
MOVL C00582 V=800.0 PL=0
MOVL C00583 V=800.0 PL=0
MOVL C00584 V=800.0 PL=0
MOVL C00585 V=800.0 PL=0
MOVL C00586 V=800.0 PL=0
MOVL C00587 V=800.0 PL=0
MOVL C00588 V=800.0 PL=0
MOVL C00589 V=800.0 PL=0
MOVL C00590 V=800.0 PL=0
MOVL C00591 V=800.0 PL=0
MOVL C00592 V=800.0 PL=0
MOVL C00593 V=800.0 PL=0
MOVL C00594 V=800.0 PL=0
MOVL C00595 V=800.0 PL=0
MOVL C00596 V=800.0 PL=0
MOVL C00597 V=800.0 PL=0
MOVL C00598 V=800.0 PL=0
MOVL C00599 V=800.0 PL=0
MOVL C00600 V=800.0 PL=0
MOVL C00601 V=800.0 PL=0
MOVL C00602 V=800.0 PL=0
MOVL C00603 V=800.0 PL=0
MOVL C00604 V=800.0 PL=0
MOVL C00605 V=800.0 PL=0
MOVL C00606 V=800.0 PL=0
MOVL C00607 V=800.0 PL=0
MOVL C00608 V=800.0 PL=0
MOVL C00609 V=800.0 PL=0
MOVL C00610 V=800.0 PL=0
MOVL C00611 V=800.0 PL=0
MOVL C00612 V=800.0 PL=0
MOVL C00613 V=800.0 PL=0
MOVL C00614 V=800.0 PL=0
MOVL C00615 V=800.0 PL=0
MOVL C00616 V=800.0 PL=0
MOVL C00617 V=800.0 PL=0
MOVL C00618 V=800.0 PL=0
MOVL C00619 V=800.0 PL=0
MOVL C00620 V=800.0 PL=0
MOVL C00621 V=800.0 PL=0
MOVL C00622 V=800.0 PL=0
MOVL C00623 V=800.0 PL=0
MOVL C00624 V=800.0 PL=0
MOVL C00625 V=800.0 PL=0
MOVL C00626 V=800.0 PL=0
MOVL C00627 V=800.0 PL=0
MOVL C00628 V=800.0 PL=0
MOVL C00629 V=800.0 PL=0
MOVL C00630 V=800.0 PL=0
MOVL C00631 V=800.0 PL=0
MOVL C00632 V=800.0 PL=0
MOVL C00633 V=800.0 PL=0
MOVL C00634 V=800.0 PL=0
MOVL C00635 V=800.0 PL=0
MOVL C00636 V=800.0 PL=0
MOVL C00637 V=800.0 PL=0
MOVL C00638 V=800.0 PL=0
MOVL C00639 V=800.0 PL=0
MOVL C00640 V=800.0 PL=0
MOVL C00641 V=800.0 PL=0
MOVL C00642 V=800.0 PL=0
MOVL C00643 V=800.0 PL=0
MOVL C00644 V=800.0 PL=0
MOVL C00645 V=800.0 PL=0
MOVL C00646 V=800.0 PL=0
MOVL C00647 V=800.0 PL=0
MOVL C00648 V=800.0 PL=0
MOVL C00649 V=800.0 PL=0
MOVL C00650 V=800.0 PL=0
MOVL C00651 V=800.0 PL=0
MOVL C00652 V=800.0 PL=0
MOVL C00653 V=800.0 PL=0
MOVL C00654 V=800.0 PL=0
MOVL C00655 V=800.0 PL=0
MOVL C00656 V=800.0 PL=0
MOVL C00657 V=800.0 PL=0
MOVL C00658 V=800.0 PL=0
MOVL C00659 V=800.0 PL=0
MOVL C00660 V=800.0 PL=0
MOVL C00661 V=800.0 PL=0
MOVL C00662 V=800.0 PL=0
MOVL C00663 V=800.0 PL=0
MOVL C00664 V=800.0 PL=0
MOVL C00665 V=800.0 PL=0
MOVL C00666 V=800.0 PL=0
MOVL C00667 V=800.0 PL=0
MOVL C00668 V=800.0 PL=0
MOVL C00669 V=800.0 PL=0
MOVL C00670 V=800.0 PL=0
MOVL C00671 V=800.0 PL=0
MOVL C00672 V=800.0 PL=0
MOVL C00673 V=800.0 PL=0
MOVL C00674 V=800.0 PL=0
MOVL C00675 V=800.0 PL=0
MOVL C00676 V=800.0 PL=0
MOVL C00677 V=800.0 PL=0
MOVL C00678 V=800.0 PL=0
MOVL C00679 V=800.0 PL=0
MOVL C00680 V=800.0 PL=0
MOVL C00681 V=800.0 PL=0
MOVL C00682 V=800.0 PL=0
MOVL C00683 V=800.0 PL=0
MOVL C00684 V=800.0 PL=0
MOVL C00685 V=800.0 PL=0
MOVL C00686 V=800.0 PL=0
MOVL C00687 V=800.0 PL=0
MOVL C00688 V=800.0 PL=0
MOVL C00689 V=800.0 PL=0
MOVL C00690 V=800.0 PL=0
MOVL C00691 V=800.0 PL=0
MOVL C00692 V=800.0 PL=0
MOVL C00693 V=800.0 PL=0
MOVL C00694 V=800.0 PL=0
MOVL C00695 V=800.0 PL=0
MOVL C00696 V=800.0 PL=0
MOVL C00697 V=800.0 PL=0
MOVL C00698 V=800.0 PL=0
MOVL C00699 V=800.0 PL=0
MOVL C00700 V=800.0 PL=0
MOVL C00701 V=800.0 PL=0
MOVL C00702 V=800.0 PL=0
MOVL C00703 V=800.0 PL=0
MOVL C00704 V=800.0 PL=0
MOVL C00705 V=800.0 PL=0
MOVL C00706 V=800.0 PL=0
MOVL C00707 V=800.0 PL=0
MOVL C00708 V=800.0 PL=0
MOVL C00709 V=800.0 PL=0
MOVL C00710 V=800.0 PL=0
MOVL C00711 V=800.0 PL=0
MOVL C00712 V=800.0 PL=0
MOVL C00713 V=800.0 PL=0
MOVL C00714 V=800.0 PL=0
MOVL C00715 V=800.0 PL=0
MOVL C00716 V=800.0 PL=0
MOVL C00717 V=800.0 PL=0
MOVL C00718 V=800.0 PL=0
MOVL C00719 V=800.0 PL=0
MOVL C00720 V=800.0 PL=0
MOVL C00721 V=800.0 PL=0
MOVL C00722 V=800.0 PL=0
MOVL C00723 V=800.0 PL=0
MOVL C00724 V=800.0 PL=0
MOVL C00725 V=800.0 PL=0
MOVL C00726 V=800.0 PL=0
MOVL C00727 V=800.0 PL=0
MOVL C00728 V=800.0 PL=0
MOVL C00729 V=800.0 PL=0
MOVL C00730 V=800.0 PL=0
MOVL C00731 V=800.0 PL=0
MOVL C00732 V=800.0 PL=0
MOVL C00733 V=800.0 PL=0
MOVL C00734 V=800.0 PL=0
MOVL C00735 V=800.0 PL=0
MOVL C00736 V=800.0 PL=0
MOVL C00737 V=800.0 PL=0
MOVL C00738 V=800.0 PL=0
MOVL C00739 V=800.0 PL=0
MOVL C00740 V=800.0 PL=0
MOVL C00741 V=800.0 PL=0
MOVL C00742 V=800.0 PL=0
MOVL C00743 V=800.0 PL=0
MOVL C00744 V=800.0 PL=0
MOVL C00745 V=800.0 PL=0
MOVL C00746 V=800.0 PL=0
MOVL C00747 V=800.0 PL=0
MOVL C00748 V=800.0 PL=0
MOVL C00749 V=800.0 PL=0
MOVL C00750 V=800.0 PL=0
MOVL C00751 V=800.0 PL=0
MOVL C00752 V=800.0 PL=0
MOVL C00753 V=800.0 PL=0
MOVL C00754 V=800.0 PL=0
MOVL C00755 V=800.0 PL=0
MOVL C00756 V=800.0 PL=0
MOVL C00757 V=800.0 PL=0
MOVL C00758 V=800.0 PL=0
MOVL C00759 V=800.0 PL=0
MOVL C00760 V=800.0 PL=0
MOVL C00761 V=800.0 PL=0
MOVL C00762 V=800.0 PL=0
MOVL C00763 V=800.0 PL=0
MOVL C00764 V=800.0 PL=0
MOVL C00765 V=800.0 PL=0
MOVL C00766 V=800.0 PL=0
MOVL C00767 V=800.0 PL=0
MOVL C00768 V=800.0 PL=0
MOVL C00769 V=800.0 PL=0
MOVL C00770 V=800.0 PL=0
MOVL C00771 V=800.0 PL=0
MOVL C00772 V=800.0 PL=0
MOVL C00773 V=800.0 PL=0
MOVL C00774 V=800.0 PL=0
MOVL C00775 V=800.0 PL=0
MOVL C00776 V=800.0 PL=0
MOVL C00777 V=800.0 PL=0
MOVL C00778 V=800.0 PL=0
MOVL C00779 V=800.0 PL=0
MOVL C00780 V=800.0 PL=0
MOVL C00781 V=800.0 PL=0
MOVL C00782 V=800.0 PL=0
MOVL C00783 V=800.0 PL=0
MOVL C00784 V=800.0 PL=0
MOVL C00785 V=800.0 PL=0
MOVL C00786 V=800.0 PL=0
MOVL C00787 V=800.0 PL=0
MOVL C00788 V=800.0 PL=0
MOVL C00789 V=800.0 PL=0
MOVL C00790 V=800.0 PL=0
MOVL C00791 V=800.0 PL=0
MOVL C00792 V=800.0 PL=0
MOVL C00793 V=800.0 PL=0
MOVL C00794 V=800.0 PL=0
MOVL C00795 V=800.0 PL=0
MOVL C00796 V=800.0 PL=0
MOVL C00797 V=800.0 PL=0
MOVL C00798 V=800.0 PL=0
MOVL C00799 V=800.0 PL=0
MOVL C00800 V=800.0 PL=0
MOVL C00801 V=800.0 PL=0
MOVL C00802 V=800.0 PL=0
MOVL C00803 V=800.0 PL=0
MOVL C00804 V=800.0 PL=0
MOVL C00805 V=800.0 PL=0
MOVL C00806 V=800.0 PL=0
MOVL C00807 V=800.0 PL=0
MOVL C00808 V=800.0 PL=0
MOVL C00809 V=800.0 PL=0
MOVL C00810 V=800.0 PL=0
MOVL C00811 V=800.0 PL=0
MOVL C00812 V=800.0 PL=0
MOVL C00813 V=800.0 PL=0
MOVL C00814 V=800.0 PL=0
MOVL C00815 V=800.0 PL=0
MOVL C00816 V=800.0 PL=0
MOVL C00817 V=800.0 PL=0
MOVL C00818 V=800.0 PL=0
MOVL C00819 V=800.0 PL=0
MOVL C00820 V=800.0 PL=0
MOVL C00821 V=800.0 PL=0
MOVL C00822 V=800.0 PL=0
MOVL C00823 V=800.0 PL=0
MOVL C00824 V=800.0 PL=0
MOVL C00825 V=800.0 PL=0
MOVL C00826 V=800.0 PL=0
MOVL C00827 V=800.0 PL=0
MOVL C00828 V=800.0 PL=0
MOVL C00829 V=800.0 PL=0
MOVL C00830 V=800.0 PL=0
MOVL C00831 V=800.0 PL=0
MOVL C00832 V=800.0 PL=0
MOVL C00833 V=800.0 PL=0
MOVL C00834 V=800.0 PL=0
MOVL C00835 V=800.0 PL=0
MOVL C00836 V=800.0 PL=0
MOVL C00837 V=800.0 PL=0
MOVL C00838 V=800.0 PL=0
MOVL C00839 V=800.0 PL=0
MOVL C00840 V=800.0 PL=0
MOVL C00841 V=800.0 PL=0
MOVL C00842 V=800.0 PL=0
MOVL C00843 V=800.0 PL=0
MOVL C00844 V=800.0 PL=0
MOVL C00845 V=800.0 PL=0
MOVL C00846 V=800.0 PL=0
MOVL C00847 V=800.0 PL=0
MOVL C00848 V=800.0 PL=0
MOVL C00849 V=800.0 PL=0
MOVL C00850 V=800.0 PL=0
MOVL C00851 V=800.0 PL=0
MOVL C00852 V=800.0 PL=0
MOVL C00853 V=800.0 PL=0
MOVL C00854 V=800.0 PL=0
MOVL C00855 V=800.0 PL=0
MOVL C00856 V=800.0 PL=0
MOVL C00857 V=800.0 PL=0
MOVL C00858 V=800.0 PL=0
MOVL C00859 V=800.0 PL=0
MOVL C00860 V=800.0 PL=0
MOVL C00861 V=800.0 PL=0
MOVL C00862 V=800.0 PL=0
MOVL C00863 V=800.0 PL=0
MOVL C00864 V=800.0 PL=0
MOVL C00865 V=800.0 PL=0
MOVL C00866 V=800.0 PL=0
MOVL C00867 V=800.0 PL=0
MOVL C00868 V=800.0 PL=0
MOVL C00869 V=800.0 PL=0
MOVL C00870 V=800.0 PL=0
MOVL C00871 V=800.0 PL=0
MOVL C00872 V=800.0 PL=0
MOVL C00873 V=800.0 PL=0
MOVL C00874 V=800.0 PL=0
MOVL C00875 V=800.0 PL=0
MOVL C00876 V=800.0 PL=0
MOVL C00877 V=800.0 PL=0
MOVL C00878 V=800.0 PL=0
MOVL C00879 V=800.0 PL=0
MOVL C00880 V=800.0 PL=0
MOVL C00881 V=800.0 PL=0
MOVL C00882 V=800.0 PL=0
MOVL C00883 V=800.0 PL=0
MOVL C00884 V=800.0 PL=0
MOVL C00885 V=800.0 PL=0
MOVL C00886 V=800.0 PL=0
MOVL C00887 V=800.0 PL=0
MOVL C00888 V=800.0 PL=0
MOVL C00889 V=800.0 PL=0
MOVL C00890 V=800.0 PL=0
MOVL C00891 V=800.0 PL=0
MOVL C00892 V=800.0 PL=0
MOVL C00893 V=800.0 PL=0
MOVL C00894 V=800.0 PL=0
MOVL C00895 V=800.0 PL=0
MOVL C00896 V=800.0 PL=0
MOVL C00897 V=800.0 PL=0
MOVL C00898 V=800.0 PL=0
MOVL C00899 V=800.0 PL=0
MOVL C00900 V=800.0 PL=0
MOVL C00901 V=800.0 PL=0
MOVL C00902 V=800.0 PL=0
MOVL C00903 V=800.0 PL=0
MOVL C00904 V=800.0 PL=0
MOVL C00905 V=800.0 PL=0
MOVL C00906 V=800.0 PL=0
MOVL C00907 V=800.0 PL=0
MOVL C00908 V=800.0 PL=0
MOVL C00909 V=800.0 PL=0
MOVL C00910 V=800.0 PL=0
MOVL C00911 V=800.0 PL=0
MOVL C00912 V=800.0 PL=0
MOVL C00913 V=800.0 PL=0
MOVL C00914 V=800.0 PL=0
MOVL C00915 V=800.0 PL=0
MOVL C00916 V=800.0 PL=0
MOVL C00917 V=800.0 PL=0
MOVL C00918 V=800.0 PL=0
MOVL C00919 V=800.0 PL=0
MOVL C00920 V=800.0 PL=0
MOVL C00921 V=800.0 PL=0
MOVL C00922 V=800.0 PL=0
MOVL C00923 V=800.0 PL=0
MOVL C00924 V=800.0 PL=0
MOVL C00925 V=800.0 PL=0
MOVL C00926 V=800.0 PL=0
MOVL C00927 V=800.0 PL=0
MOVL C00928 V=800.0 PL=0
MOVL C00929 V=800.0 PL=0
MOVL C00930 V=800.0 PL=0
MOVL C00931 V=800.0 PL=0
MOVL C00932 V=800.0 PL=0
MOVL C00933 V=800.0 PL=0
MOVL C00934 V=800.0 PL=0
MOVL C00935 V=800.0 PL=0
MOVL C00936 V=800.0 PL=0
MOVL C00937 V=800.0 PL=0
MOVL C00938 V=800.0 PL=0
MOVL C00939 V=800.0 PL=0
MOVL C00940 V=800.0 PL=0
MOVL C00941 V=800.0 PL=0
MOVL C00942 V=800.0 PL=0
MOVL C00943 V=800.0 PL=0
MOVL C00944 V=800.0 PL=0
MOVL C00945 V=800.0 PL=0
MOVL C00946 V=800.0 PL=0
MOVL C00947 V=800.0 PL=0
MOVL C00948 V=800.0 PL=0
MOVL C00949 V=800.0 PL=0
MOVL C00950 V=800.0 PL=0
MOVL C00951 V=800.0 PL=0
MOVL C00952 V=800.0 PL=0
MOVL C00953 V=800.0 PL=0
MOVL C00954 V=800.0 PL=0
MOVL C00955 V=800.0 PL=0
MOVL C00956 V=800.0 PL=0
MOVL C00957 V=800.0 PL=0
MOVL C00958 V=800.0 PL=0
MOVL C00959 V=800.0 PL=0
MOVL C00960 V=800.0 PL=0
MOVL C00961 V=800.0 PL=0
MOVL C00962 V=800.0 PL=0
MOVL C00963 V=800.0 PL=0
MOVL C00964 V=800.0 PL=0
MOVL C00965 V=800.0 PL=0
MOVL C00966 V=800.0 PL=0
MOVL C00967 V=800.0 PL=0
MOVL C00968 V=800.0 PL=0
MOVL C00969 V=800.0 PL=0
MOVL C00970 V=800.0 PL=0
MOVL C00971 V=800.0 PL=0
MOVL C00972 V=800.0 PL=0
MOVL C00973 V=800.0 PL=0
MOVL C00974 V=800.0 PL=0
MOVL C00975 V=800.0 PL=0
MOVL C00976 V=800.0 PL=0
MOVL C00977 V=800.0 PL=0
MOVL C00978 V=800.0 PL=0
MOVL C00979 V=800.0 PL=0
MOVL C00980 V=800.0 PL=0
MOVL C00981 V=800.0 PL=0
MOVL C00982 V=800.0 PL=0
MOVL C00983 V=800.0 PL=0
MOVL C00984 V=800.0 PL=0
MOVL C00985 V=800.0 PL=0
MOVL C00986 V=800.0 PL=0
MOVL C00987 V=800.0 PL=0
MOVL C00988 V=800.0 PL=0
MOVL C00989 V=800.0 PL=0
MOVL C00990 V=800.0 PL=0
MOVL C00991 V=800.0 PL=0
MOVL C00992 V=800.0 PL=0
MOVL C00993 V=800.0 PL=0
MOVL C00994 V=800.0 PL=0
MOVL C00995 V=800.0 PL=0
MOVL C00996 V=800.0 PL=0
MOVL C00997 V=800.0 PL=0
MOVL C00998 V=800.0 PL=0
MOVL C00999 V=800.0 PL=0
MOVL C01000 V=800.0 PL=0
MOVL C01001 V=800.0 PL=0
MOVL C01002 V=800.0 PL=0
MOVL C01003 V=800.0 PL=0
MOVL C01004 V=800.0 PL=0
MOVL C01005 V=800.0 PL=0
MOVL C01006 V=800.0 PL=0
MOVL C01007 V=800.0 PL=0
MOVL C01008 V=800.0 PL=0
MOVL C01009 V=800.0 PL=0
MOVL C01010 V=800.0 PL=0
MOVL C01011 V=800.0 PL=0
MOVL C01012 V=800.0 PL=0
MOVL C01013 V=800.0 PL=0
MOVL C01014 V=800.0 PL=0
MOVL C01015 V=800.0 PL=0
MOVL C01016 V=800.0 PL=0
MOVL C01017 V=800.0 PL=0
MOVL C01018 V=800.0 PL=0
MOVL C01019 V=800.0 PL=0
MOVL C01020 V=800.0 PL=0
MOVL C01021 V=800.0 PL=0
MOVL C01022 V=800.0 PL=0
MOVL C01023 V=800.0 PL=0
MOVL C01024 V=800.0 PL=0
MOVL C01025 V=800.0 PL=0
MOVL C01026 V=800.0 PL=0
MOVL C01027 V=800.0 PL=0
MOVL C01028 V=800.0 PL=0
MOVL C01029 V=800.0 PL=0
MOVL C01030 V=800.0 PL=0
MOVL C01031 V=800.0 PL=0
MOVL C01032 V=800.0 PL=0
MOVL C01033 V=800.0 PL=0
MOVL C01034 V=800.0 PL=0
MOVL C01035 V=800.0 PL=0
MOVL C01036 V=800.0 PL=0
MOVL C01037 V=800.0 PL=0
MOVL C01038 V=800.0 PL=0
MOVL C01039 V=800.0 PL=0
MOVL C01040 V=800.0 PL=0
MOVL C01041 V=800.0 PL=0
MOVL C01042 V=800.0 PL=0
MOVL C01043 V=800.0 PL=0
MOVL C01044 V=800.0 PL=0
MOVL C01045 V=800.0 PL=0
MOVL C01046 V=800.0 PL=0
MOVL C01047 V=800.0 PL=0
MOVL C01048 V=800.0 PL=0
MOVL C01049 V=800.0 PL=0
MOVL C01050 V=800.0 PL=0
MOVL C01051 V=800.0 PL=0
MOVL C01052 V=800.0 PL=0
MOVL C01053 V=800.0 PL=0
MOVL C01054 V=800.0 PL=0
MOVL C01055 V=800.0 PL=0
MOVL C01056 V=800.0 PL=0
MOVL C01057 V=800.0 PL=0
MOVL C01058 V=800.0 PL=0
MOVL C01059 V=800.0 PL=0
MOVL C01060 V=800.0 PL=0
MOVL C01061 V=800.0 PL=0
MOVL C01062 V=800.0 PL=0
MOVL C01063 V=800.0 PL=0
MOVL C01064 V=800.0 PL=0
MOVL C01065 V=800.0 PL=0
MOVL C01066 V=800.0 PL=0
MOVL C01067 V=800.0 PL=0
MOVL C01068 V=800.0 PL=0
MOVL C01069 V=800.0 PL=0
MOVL C01070 V=800.0 PL=0
MOVL C01071 V=800.0 PL=0
MOVL C01072 V=800.0 PL=0
MOVL C01073 V=800.0 PL=0
MOVL C01074 V=800.0 PL=0
MOVL C01075 V=800.0 PL=0
MOVL C01076 V=800.0 PL=0
MOVL C01077 V=800.0 PL=0
MOVL C01078 V=800.0 PL=0
MOVL C01079 V=800.0 PL=0
MOVL C01080 V=800.0 PL=0
MOVL C01081 V=800.0 PL=0
MOVL C01082 V=800.0 PL=0
MOVL C01083 V=800.0 PL=0
MOVL C01084 V=800.0 PL=0
MOVL C01085 V=800.0 PL=0
MOVL C01086 V=800.0 PL=0
MOVL C01087 V=800.0 PL=0
MOVL C01088 V=800.0 PL=0
MOVL C01089 V=800.0 PL=0
MOVL C01090 V=800.0 PL=0
MOVL C01091 V=800.0 PL=0
MOVL C01092 V=800.0 PL=0
MOVL C01093 V=800.0 PL=0
MOVL C01094 V=800.0 PL=0
MOVL C01095 V=800.0 PL=0
MOVL C01096 V=800.0 PL=0
MOVL C01097 V=800.0 PL=0
MOVL C01098 V=800.0 PL=0
MOVL C01099 V=800.0 PL=0
MOVL C01100 V=800.0 PL=0
MOVL C01101 V=800.0 PL=0
MOVL C01102 V=800.0 PL=0
MOVL C01103 V=800.0 PL=0
MOVL C01104 V=800.0 PL=0
MOVL C01105 V=800.0 PL=0
MOVL C01106 V=800.0 PL=0
MOVL C01107 V=800.0 PL=0
MOVL C01108 V=800.0 PL=0
MOVL C01109 V=800.0 PL=0
MOVL C01110 V=800.0 PL=0
MOVL C01111 V=800.0 PL=0
MOVL C01112 V=800.0 PL=0
MOVL C01113 V=800.0 PL=0
MOVL C01114 V=800.0 PL=0
MOVL C01115 V=800.0 PL=0
MOVL C01116 V=800.0 PL=0
MOVL C01117 V=800.0 PL=0
MOVL C01118 V=800.0 PL=0
MOVL C01119 V=800.0 PL=0
MOVL C01120 V=800.0 PL=0
MOVL C01121 V=800.0 PL=0
MOVL C01122 V=800.0 PL=0
MOVL C01123 V=800.0 PL=0
MOVL C01124 V=800.0 PL=0
MOVL C01125 V=800.0 PL=0
MOVL C01126 V=800.0 PL=0
MOVL C01127 V=800.0 PL=0
MOVL C01128 V=800.0 PL=0
MOVL C01129 V=800.0 PL=0
MOVL C01130 V=800.0 PL=0
MOVL C01131 V=800.0 PL=0
MOVL C01132 V=800.0 PL=0
MOVL C01133 V=800.0 PL=0
MOVL C01134 V=800.0 PL=0
MOVL C01135 V=800.0 PL=0
MOVL C01136 V=800.0 PL=0
MOVL C01137 V=800.0 PL=0
MOVL C01138 V=800.0 PL=0
MOVL C01139 V=800.0 PL=0
MOVL C01140 V=800.0 PL=0
MOVL C01141 V=800.0 PL=0
MOVL C01142 V=800.0 PL=0
MOVL C01143 V=800.0 PL=0
MOVL C01144 V=800.0 PL=0
MOVL C01145 V=800.0 PL=0
MOVL C01146 V=800.0 PL=0
MOVL C01147 V=800.0 PL=0
MOVL C01148 V=800.0 PL=0
MOVL C01149 V=800.0 PL=0
MOVL C01150 V=800.0 PL=0
MOVL C01151 V=800.0 PL=0
MOVL C01152 V=800.0 PL=0
MOVL C01153 V=800.0 PL=0
MOVL C01154 V=800.0 PL=0
MOVL C01155 V=800.0 PL=0
MOVL C01156 V=800.0 PL=0
MOVL C01157 V=800.0 PL=0
MOVL C01158 V=800.0 PL=0
MOVL C01159 V=800.0 PL=0
MOVL C01160 V=800.0 PL=0
MOVL C01161 V=800.0 PL=0
MOVL C01162 V=800.0 PL=0
MOVL C01163 V=800.0 PL=0
MOVL C01164 V=800.0 PL=0
MOVL C01165 V=800.0 PL=0
MOVL C01166 V=800.0 PL=0
MOVL C01167 V=800.0 PL=0
MOVL C01168 V=800.0 PL=0
MOVL C01169 V=800.0 PL=0
MOVL C01170 V=800.0 PL=0
MOVL C01171 V=800.0 PL=0
MOVL C01172 V=800.0 PL=0
MOVL C01173 V=800.0 PL=0
MOVL C01174 V=800.0 PL=0
MOVL C01175 V=800.0 PL=0
MOVL C01176 V=800.0 PL=0
MOVL C01177 V=800.0 PL=0
MOVL C01178 V=800.0 PL=0
MOVL C01179 V=800.0 PL=0
MOVL C01180 V=800.0 PL=0
MOVL C01181 V=800.0 PL=0
MOVL C01182 V=800.0 PL=0
MOVL C01183 V=800.0 PL=0
MOVL C01184 V=800.0 PL=0
MOVL C01185 V=800.0 PL=0
MOVL C01186 V=800.0 PL=0
MOVL C01187 V=800.0 PL=0
MOVL C01188 V=800.0 PL=0
MOVL C01189 V=800.0 PL=0
MOVL C01190 V=800.0 PL=0
MOVL C01191 V=800.0 PL=0
MOVL C01192 V=800.0 PL=0
MOVL C01193 V=800.0 PL=0
MOVL C01194 V=800.0 PL=0
MOVL C01195 V=800.0 PL=0
MOVL C01196 V=800.0 PL=0
MOVL C01197 V=800.0 PL=0
MOVL C01198 V=800.0 PL=0
MOVL C01199 V=800.0 PL=0
MOVL C01200 V=800.0 PL=0
MOVL C01201 V=800.0 PL=0
MOVL C01202 V=800.0 PL=0
MOVL C01203 V=800.0 PL=0
MOVL C01204 V=800.0 PL=0
MOVL C01205 V=800.0 PL=0
MOVL C01206 V=800.0 PL=0
MOVL C01207 V=800.0 PL=0
MOVL C01208 V=800.0 PL=0
MOVL C01209 V=800.0 PL=0
MOVL C01210 V=800.0 PL=0
MOVL C01211 V=800.0 PL=0
MOVL C01212 V=800.0 PL=0
MOVL C01213 V=800.0 PL=0
MOVL C01214 V=800.0 PL=0
MOVL C01215 V=800.0 PL=0
MOVL C01216 V=800.0 PL=0
MOVL C01217 V=800.0 PL=0
MOVL C01218 V=800.0 PL=0
MOVL C01219 V=800.0 PL=0
MOVL C01220 V=800.0 PL=0
MOVL C01221 V=800.0 PL=0
MOVL C01222 V=800.0 PL=0
MOVL C01223 V=800.0 PL=0
MOVL C01224 V=800.0 PL=0
MOVL C01225 V=800.0 PL=0
MOVL C01226 V=800.0 PL=0
MOVL C01227 V=800.0 PL=0
MOVL C01228 V=800.0 PL=0
MOVL C01229 V=800.0 PL=0
MOVL C01230 V=800.0 PL=0
MOVL C01231 V=800.0 PL=0
MOVL C01232 V=800.0 PL=0
MOVL C01233 V=800.0 PL=0
MOVL C01234 V=800.0 PL=0
MOVL C01235 V=800.0 PL=0
MOVL C01236 V=800.0 PL=0
MOVL C01237 V=800.0 PL=0
MOVL C01238 V=800.0 PL=0
MOVL C01239 V=800.0 PL=0
MOVL C01240 V=800.0 PL=0
MOVL C01241 V=800.0 PL=0
MOVL C01242 V=800.0 PL=0
MOVL C01243 V=800.0 PL=0
MOVL C01244 V=800.0 PL=0
MOVL C01245 V=800.0 PL=0
MOVL C01246 V=800.0 PL=0
MOVL C01247 V=800.0 PL=0
MOVL C01248 V=800.0 PL=0
MOVL C01249 V=800.0 PL=0
MOVL C01250 V=800.0 PL=0
MOVL C01251 V=800.0 PL=0
MOVL C01252 V=800.0 PL=0
MOVL C01253 V=800.0 PL=0
MOVL C01254 V=800.0 PL=0
MOVL C01255 V=800.0 PL=0
MOVL C01256 V=800.0 PL=0
MOVL C01257 V=800.0 PL=0
MOVL C01258 V=800.0 PL=0
MOVL C01259 V=800.0 PL=0
MOVL C01260 V=800.0 PL=0
MOVL C01261 V=800.0 PL=0
MOVL C01262 V=800.0 PL=0
MOVL C01263 V=800.0 PL=0
MOVL C01264 V=800.0 PL=0
MOVL C01265 V=800.0 PL=0
MOVL C01266 V=800.0 PL=0
MOVL C01267 V=800.0 PL=0
MOVL C01268 V=800.0 PL=0
MOVL C01269 V=800.0 PL=0
MOVL C01270 V=800.0 PL=0
MOVL C01271 V=800.0 PL=0
MOVL C01272 V=800.0 PL=0
MOVL C01273 V=800.0 PL=0
MOVL C01274 V=800.0 PL=0
MOVL C01275 V=800.0 PL=0
MOVL C01276 V=800.0 PL=0
MOVL C01277 V=800.0 PL=0
MOVL C01278 V=800.0 PL=0
MOVL C01279 V=800.0 PL=0
MOVL C01280 V=800.0 PL=0
MOVL C01281 V=800.0 PL=0
MOVL C01282 V=800.0 PL=0
MOVL C01283 V=800.0 PL=0
MOVL C01284 V=800.0 PL=0
MOVL C01285 V=800.0 PL=0
MOVL C01286 V=800.0 PL=0
MOVL C01287 V=800.0 PL=0
MOVL C01288 V=800.0 PL=0
MOVL C01289 V=800.0 PL=0
MOVL C01290 V=800.0 PL=0
MOVL C01291 V=800.0 PL=0
MOVL C01292 V=800.0 PL=0
MOVL C01293 V=800.0 PL=0
MOVL C01294 V=800.0 PL=0
MOVL C01295 V=800.0 PL=0
MOVL C01296 V=800.0 PL=0
MOVL C01297 V=800.0 PL=0
MOVL C01298 V=800.0 PL=0
MOVL C01299 V=800.0 PL=0
MOVL C01300 V=800.0 PL=0
MOVL C01301 V=800.0 PL=0
MOVL C01302 V=800.0 PL=0
MOVL C01303 V=800.0 PL=0
MOVL C01304 V=800.0 PL=0
MOVL C01305 V=800.0 PL=0
MOVL C01306 V=800.0 PL=0
MOVL C01307 V=800.0 PL=0
MOVL C01308 V=800.0 PL=0
MOVL C01309 V=800.0 PL=0
MOVL C01310 V=800.0 PL=0
MOVL C01311 V=800.0 PL=0
MOVL C01312 V=800.0 PL=0
MOVL C01313 V=800.0 PL=0
MOVL C01314 V=800.0 PL=0
MOVL C01315 V=800.0 PL=0
MOVL C01316 V=800.0 PL=0
MOVL C01317 V=800.0 PL=0
MOVL C01318 V=800.0 PL=0
MOVL C01319 V=800.0 PL=0
MOVL C01320 V=800.0 PL=0
MOVL C01321 V=800.0 PL=0
MOVL C01322 V=800.0 PL=0
MOVL C01323 V=800.0 PL=0
MOVL C01324 V=800.0 PL=0
MOVL C01325 V=800.0 PL=0
MOVL C01326 V=800.0 PL=0
MOVL C01327 V=800.0 PL=0
MOVL C01328 V=800.0 PL=0
MOVL C01329 V=800.0 PL=0
MOVL C01330 V=800.0 PL=0
MOVL C01331 V=800.0 PL=0
MOVL C01332 V=800.0 PL=0
MOVL C01333 V=800.0 PL=0
MOVL C01334 V=800.0 PL=0
MOVL C01335 V=800.0 PL=0
MOVL C01336 V=800.0 PL=0
MOVL C01337 V=800.0 PL=0
MOVL C01338 V=800.0 PL=0
MOVL C01339 V=800.0 PL=0
MOVL C01340 V=800.0 PL=0
MOVL C01341 V=800.0 PL=0
MOVL C01342 V=800.0 PL=0
MOVL C01343 V=800.0 PL=0
MOVL C01344 V=800.0 PL=0
MOVL C01345 V=800.0 PL=0
MOVL C01346 V=800.0 PL=0
MOVL C01347 V=800.0 PL=0
MOVL C01348 V=800.0 PL=0
MOVL C01349 V=800.0 PL=0
MOVL C01350 V=800.0 PL=0
MOVL C01351 V=800.0 PL=0
MOVL C01352 V=800.0 PL=0
MOVL C01353 V=800.0 PL=0
MOVL C01354 V=800.0 PL=0
MOVL C01355 V=800.0 PL=0
MOVL C01356 V=800.0 PL=0
MOVL C01357 V=800.0 PL=0
MOVL C01358 V=800.0 PL=0
MOVL C01359 V=800.0 PL=0
MOVL C01360 V=800.0 PL=0
MOVL C01361 V=800.0 PL=0
MOVL C01362 V=800.0 PL=0
MOVL C01363 V=800.0 PL=0
MOVL C01364 V=800.0 PL=0
MOVL C01365 V=800.0 PL=0
MOVL C01366 V=800.0 PL=0
MOVL C01367 V=800.0 PL=0
MOVL C01368 V=800.0 PL=0
MOVL C01369 V=800.0 PL=0
MOVL C01370 V=800.0 PL=0
MOVL C01371 V=800.0 PL=0
MOVL C01372 V=800.0 PL=0
MOVL C01373 V=800.0 PL=0
MOVL C01374 V=800.0 PL=0
MOVL C01375 V=800.0 PL=0
MOVL C01376 V=800.0 PL=0
MOVL C01377 V=800.0 PL=0
MOVL C01378 V=800.0 PL=0
MOVL C01379 V=800.0 PL=0
MOVL C01380 V=800.0 PL=0
MOVL C01381 V=800.0 PL=0
MOVL C01382 V=800.0 PL=0
MOVL C01383 V=800.0 PL=0
MOVL C01384 V=800.0 PL=0
MOVL C01385 V=800.0 PL=0
MOVL C01386 V=800.0 PL=0
MOVL C01387 V=800.0 PL=0
MOVL C01388 V=800.0 PL=0
MOVL C01389 V=800.0 PL=0
MOVL C01390 V=800.0 PL=0
MOVL C01391 V=800.0 PL=0
MOVL C01392 V=800.0 PL=0
MOVL C01393 V=800.0 PL=0
MOVL C01394 V=800.0 PL=0
MOVL C01395 V=800.0 PL=0
MOVL C01396 V=800.0 PL=0
MOVL C01397 V=800.0 PL=0
MOVL C01398 V=800.0 PL=0
MOVL C01399 V=800.0 PL=0
MOVL C01400 V=800.0 PL=0
MOVL C01401 V=800.0 PL=0
MOVL C01402 V=800.0 PL=0
MOVL C01403 V=800.0 PL=0
MOVL C01404 V=800.0 PL=0
MOVL C01405 V=800.0 PL=0
MOVL C01406 V=800.0 PL=0
MOVL C01407 V=800.0 PL=0
MOVL C01408 V=800.0 PL=0
MOVL C01409 V=800.0 PL=0
MOVL C01410 V=800.0 PL=0
MOVL C01411 V=800.0 PL=0
MOVL C01412 V=800.0 PL=0
MOVL C01413 V=800.0 PL=0
MOVL C01414 V=800.0 PL=0
MOVL C01415 V=800.0 PL=0
MOVL C01416 V=800.0 PL=0
MOVL C01417 V=800.0 PL=0
MOVL C01418 V=800.0 PL=0
MOVL C01419 V=800.0 PL=0
MOVL C01420 V=800.0 PL=0
MOVL C01421 V=800.0 PL=0
MOVL C01422 V=800.0 PL=0
MOVL C01423 V=800.0 PL=0
MOVL C01424 V=800.0 PL=0
MOVL C01425 V=800.0 PL=0
MOVL C01426 V=800.0 PL=0
MOVL C01427 V=800.0 PL=0
MOVL C01428 V=800.0 PL=0
MOVL C01429 V=800.0 PL=0
MOVL C01430 V=800.0 PL=0
MOVL C01431 V=800.0 PL=0
MOVL C01432 V=800.0 PL=0
MOVL C01433 V=800.0 PL=0
MOVL C01434 V=800.0 PL=0
MOVL C01435 V=800.0 PL=0
MOVL C01436 V=800.0 PL=0
MOVL C01437 V=800.0 PL=0
MOVL C01438 V=800.0 PL=0
MOVL C01439 V=800.0 PL=0
MOVL C01440 V=800.0 PL=0
MOVL C01441 V=800.0 PL=0
MOVL C01442 V=800.0 PL=0
MOVL C01443 V=800.0 PL=0
MOVL C01444 V=800.0 PL=0
MOVL C01445 V=800.0 PL=0
MOVL C01446 V=800.0 PL=0
MOVL C01447 V=800.0 PL=0
MOVL C01448 V=800.0 PL=0
MOVL C01449 V=800.0 PL=0
MOVL C01450 V=800.0 PL=0
MOVL C01451 V=800.0 PL=0
MOVL C01452 V=800.0 PL=0
MOVL C01453 V=800.0 PL=0
MOVL C01454 V=800.0 PL=0
MOVL C01455 V=800.0 PL=0
MOVL C01456 V=800.0 PL=0
MOVL C01457 V=800.0 PL=0
MOVL C01458 V=800.0 PL=0
MOVL C01459 V=800.0 PL=0
MOVL C01460 V=800.0 PL=0
MOVL C01461 V=800.0 PL=0
MOVL C01462 V=800.0 PL=0
MOVL C01463 V=800.0 PL=0
MOVL C01464 V=800.0 PL=0
MOVL C01465 V=800.0 PL=0
MOVL C01466 V=800.0 PL=0
MOVL C01467 V=800.0 PL=0
MOVL C01468 V=800.0 PL=0
MOVL C01469 V=800.0 PL=0
MOVL C01470 V=800.0 PL=0
MOVL C01471 V=800.0 PL=0
MOVL C01472 V=800.0 PL=0
MOVL C01473 V=800.0 PL=0
MOVL C01474 V=800.0 PL=0
MOVL C01475 V=800.0 PL=0
MOVL C01476 V=800.0 PL=0
MOVL C01477 V=800.0 PL=0
MOVL C01478 V=800.0 PL=0
MOVL C01479 V=800.0 PL=0
MOVL C01480 V=800.0 PL=0
MOVL C01481 V=800.0 PL=0
MOVL C01482 V=800.0 PL=0
MOVL C01483 V=800.0 PL=0
MOVL C01484 V=800.0 PL=0
MOVL C01485 V=800.0 PL=0
MOVL C01486 V=800.0 PL=0
MOVL C01487 V=800.0 PL=0
MOVL C01488 V=800.0 PL=0
MOVL C01489 V=800.0 PL=0
MOVL C01490 V=800.0 PL=0
MOVL C01491 V=800.0 PL=0
MOVL C01492 V=800.0 PL=0
MOVL C01493 V=800.0 PL=0
MOVL C01494 V=800.0 PL=0
MOVL C01495 V=800.0 PL=0
MOVL C01496 V=800.0 PL=0
MOVL C01497 V=800.0 PL=0
MOVL C01498 V=800.0 PL=0
MOVL C01499 V=800.0 PL=0
MOVL C01500 V=800.0 PL=0
MOVL C01501 V=800.0 PL=0
MOVL C01502 V=800.0 PL=0
MOVL C01503 V=800.0 PL=0
MOVL C01504 V=800.0 PL=0
MOVL C01505 V=800.0 PL=0
MOVL C01506 V=800.0 PL=0
MOVL C01507 V=800.0 PL=0
MOVL C01508 V=800.0 PL=0
MOVL C01509 V=800.0 PL=0
MOVL C01510 V=800.0 PL=0
MOVL C01511 V=800.0 PL=0
MOVL C01512 V=800.0 PL=0
MOVL C01513 V=800.0 PL=0
MOVL C01514 V=800.0 PL=0
MOVL C01515 V=800.0 PL=0
MOVL C01516 V=800.0 PL=0
MOVL C01517 V=800.0 PL=0
MOVL C01518 V=800.0 PL=0
MOVL C01519 V=800.0 PL=0
MOVL C01520 V=800.0 PL=0
MOVL C01521 V=800.0 PL=0
MOVL C01522 V=800.0 PL=0
MOVL C01523 V=800.0 PL=0
MOVL C01524 V=800.0 PL=0
MOVL C01525 V=800.0 PL=0
MOVL C01526 V=800.0 PL=0
MOVL C01527 V=800.0 PL=0
MOVL C01528 V=800.0 PL=0
MOVL C01529 V=800.0 PL=0
MOVL C01530 V=800.0 PL=0
MOVL C01531 V=800.0 PL=0
MOVL C01532 V=800.0 PL=0
MOVL C01533 V=800.0 PL=0
MOVL C01534 V=800.0 PL=0
MOVL C01535 V=800.0 PL=0
MOVL C01536 V=800.0 PL=0
MOVL C01537 V=800.0 PL=0
MOVL C01538 V=800.0 PL=0
MOVL C01539 V=800.0 PL=0
MOVL C01540 V=800.0 PL=0
MOVL C01541 V=800.0 PL=0
MOVL C01542 V=800.0 PL=0
MOVL C01543 V=800.0 PL=0
MOVL C01544 V=800.0 PL=0
MOVL C01545 V=800.0 PL=0
MOVL C01546 V=800.0 PL=0
MOVL C01547 V=800.0 PL=0
MOVL C01548 V=800.0 PL=0
MOVL C01549 V=800.0 PL=0
MOVL C01550 V=800.0 PL=0
MOVL C01551 V=800.0 PL=0
MOVL C01552 V=800.0 PL=0
MOVL C01553 V=800.0 PL=0
MOVL C01554 V=800.0 PL=0
MOVL C01555 V=800.0 PL=0
MOVL C01556 V=800.0 PL=0
MOVL C01557 V=800.0 PL=0
MOVL C01558 V=800.0 PL=0
MOVL C01559 V=800.0 PL=0
MOVL C01560 V=800.0 PL=0
MOVL C01561 V=800.0 PL=0
MOVL C01562 V=800.0 PL=0
MOVL C01563 V=800.0 PL=0
MOVL C01564 V=800.0 PL=0
MOVL C01565 V=800.0 PL=0
MOVL C01566 V=800.0 PL=0
MOVL C01567 V=800.0 PL=0
MOVL C01568 V=800.0 PL=0
MOVL C01569 V=800.0 PL=0
MOVL C01570 V=800.0 PL=0
MOVL C01571 V=800.0 PL=0
MOVL C01572 V=800.0 PL=0
MOVL C01573 V=800.0 PL=0
MOVL C01574 V=800.0 PL=0
MOVL C01575 V=800.0 PL=0
MOVL C01576 V=800.0 PL=0
MOVL C01577 V=800.0 PL=0
MOVL C01578 V=800.0 PL=0
MOVL C01579 V=800.0 PL=0
MOVL C01580 V=800.0 PL=0
MOVL C01581 V=800.0 PL=0
MOVL C01582 V=800.0 PL=0
MOVL C01583 V=800.0 PL=0
MOVL C01584 V=800.0 PL=0
MOVL C01585 V=800.0 PL=0
MOVL C01586 V=800.0 PL=0
MOVL C01587 V=800.0 PL=0
MOVL C01588 V=800.0 PL=0
MOVL C01589 V=800.0 PL=0
MOVL C01590 V=800.0 PL=0
MOVL C01591 V=800.0 PL=0
MOVL C01592 V=800.0 PL=0
MOVL C01593 V=800.0 PL=0
MOVL C01594 V=800.0 PL=0
MOVL C01595 V=800.0 PL=0
MOVL C01596 V=800.0 PL=0
MOVL C01597 V=800.0 PL=0
MOVL C01598 V=800.0 PL=0
MOVL C01599 V=800.0 PL=0
MOVL C01600 V=800.0 PL=0
MOVL C01601 V=800.0 PL=0
MOVL C01602 V=800.0 PL=0
MOVL C01603 V=800.0 PL=0
MOVL C01604 V=800.0 PL=0
MOVL C01605 V=800.0 PL=0
MOVL C01606 V=800.0 PL=0
MOVL C01607 V=800.0 PL=0
MOVL C01608 V=800.0 PL=0
MOVL C01609 V=800.0 PL=0
MOVL C01610 V=800.0 PL=0
MOVL C01611 V=800.0 PL=0
MOVL C01612 V=800.0 PL=0
MOVL C01613 V=800.0 PL=0
MOVL C01614 V=800.0 PL=0
MOVL C01615 V=800.0 PL=0
MOVL C01616 V=800.0 PL=0
MOVL C01617 V=800.0 PL=0
MOVL C01618 V=800.0 PL=0
MOVL C01619 V=800.0 PL=0
MOVL C01620 V=800.0 PL=0
MOVL C01621 V=800.0 PL=0
MOVL C01622 V=800.0 PL=0
MOVL C01623 V=800.0 PL=0
MOVL C01624 V=800.0 PL=0
MOVL C01625 V=800.0 PL=0
MOVL C01626 V=800.0 PL=0
MOVL C01627 V=800.0 PL=0
MOVL C01628 V=800.0 PL=0
MOVL C01629 V=800.0 PL=0
MOVL C01630 V=800.0 PL=0
MOVL C01631 V=800.0 PL=0
MOVL C01632 V=800.0 PL=0
MOVL C01633 V=800.0 PL=0
MOVL C01634 V=800.0 PL=0
MOVL C01635 V=800.0 PL=0
MOVL C01636 V=800.0 PL=0
MOVL C01637 V=800.0 PL=0
MOVL C01638 V=800.0 PL=0
MOVL C01639 V=800.0 PL=0
MOVL C01640 V=800.0 PL=0
MOVL C01641 V=800.0 PL=0
MOVL C01642 V=800.0 PL=0
MOVL C01643 V=800.0 PL=0
MOVL C01644 V=800.0 PL=0
MOVL C01645 V=800.0 PL=0
MOVL C01646 V=800.0 PL=0
MOVL C01647 V=800.0 PL=0
MOVL C01648 V=800.0 PL=0
MOVL C01649 V=800.0 PL=0
MOVL C01650 V=800.0 PL=0
MOVL C01651 V=800.0 PL=0
MOVL C01652 V=800.0 PL=0
MOVL C01653 V=800.0 PL=0
MOVL C01654 V=800.0 PL=0
MOVL C01655 V=800.0 PL=0
MOVL C01656 V=800.0 PL=0
MOVL C01657 V=800.0 PL=0
MOVL C01658 V=800.0 PL=0
MOVL C01659 V=800.0 PL=0
MOVL C01660 V=800.0 PL=0
MOVL C01661 V=800.0 PL=0
MOVL C01662 V=800.0 PL=0
MOVL C01663 V=800.0 PL=0
MOVL C01664 V=800.0 PL=0
MOVL C01665 V=800.0 PL=0
MOVL C01666 V=800.0 PL=0
MOVL C01667 V=800.0 PL=0
MOVL C01668 V=800.0 PL=0
MOVL C01669 V=800.0 PL=0
MOVL C01670 V=800.0 PL=0
MOVL C01671 V=800.0 PL=0
MOVL C01672 V=800.0 PL=0
MOVL C01673 V=800.0 PL=0
MOVL C01674 V=800.0 PL=0
MOVL C01675 V=800.0 PL=0
MOVL C01676 V=800.0 PL=0
MOVL C01677 V=800.0 PL=0
MOVL C01678 V=800.0 PL=0
MOVL C01679 V=800.0 PL=0
MOVL C01680 V=800.0 PL=0
MOVL C01681 V=800.0 PL=0
MOVL C01682 V=800.0 PL=0
MOVL C01683 V=800.0 PL=0
MOVL C01684 V=800.0 PL=0
MOVL C01685 V=800.0 PL=0
MOVL C01686 V=800.0 PL=0
MOVL C01687 V=800.0 PL=0
MOVL C01688 V=800.0 PL=0
MOVL C01689 V=800.0 PL=0
MOVL C01690 V=800.0 PL=0
MOVL C01691 V=800.0 PL=0
MOVL C01692 V=800.0 PL=0
MOVL C01693 V=800.0 PL=0
MOVL C01694 V=800.0 PL=0
MOVL C01695 V=800.0 PL=0
MOVL C01696 V=800.0 PL=0
MOVL C01697 V=800.0 PL=0
MOVL C01698 V=800.0 PL=0
MOVL C01699 V=800.0 PL=0
MOVL C01700 V=800.0 PL=0
MOVL C01701 V=800.0 PL=0
MOVL C01702 V=800.0 PL=0
MOVL C01703 V=800.0 PL=0
MOVL C01704 V=800.0 PL=0
MOVL C01705 V=800.0 PL=0
MOVL C01706 V=800.0 PL=0
MOVL C01707 V=800.0 PL=0
MOVL C01708 V=800.0 PL=0
MOVL C01709 V=800.0 PL=0
MOVL C01710 V=800.0 PL=0
MOVL C01711 V=800.0 PL=0
MOVL C01712 V=800.0 PL=0
MOVL C01713 V=800.0 PL=0
MOVL C01714 V=800.0 PL=0
MOVL C01715 V=800.0 PL=0
MOVL C01716 V=800.0 PL=0
MOVL C01717 V=800.0 PL=0
MOVL C01718 V=800.0 PL=0
MOVL C01719 V=800.0 PL=0
MOVL C01720 V=800.0 PL=0
MOVL C01721 V=800.0 PL=0
MOVL C01722 V=800.0 PL=0
MOVL C01723 V=800.0 PL=0
MOVL C01724 V=800.0 PL=0
MOVL C01725 V=800.0 PL=0
MOVL C01726 V=800.0 PL=0
MOVL C01727 V=800.0 PL=0
MOVL C01728 V=800.0 PL=0
MOVL C01729 V=800.0 PL=0
MOVL C01730 V=800.0 PL=0
MOVL C01731 V=800.0 PL=0
MOVL C01732 V=800.0 PL=0
MOVL C01733 V=800.0 PL=0
MOVL C01734 V=800.0 PL=0
MOVL C01735 V=800.0 PL=0
MOVL C01736 V=800.0 PL=0
MOVL C01737 V=800.0 PL=0
MOVL C01738 V=800.0 PL=0
MOVL C01739 V=800.0 PL=0
MOVL C01740 V=800.0 PL=0
MOVL C01741 V=800.0 PL=0
MOVL C01742 V=800.0 PL=0
MOVL C01743 V=800.0 PL=0
MOVL C01744 V=800.0 PL=0
MOVL C01745 V=800.0 PL=0
MOVL C01746 V=800.0 PL=0
MOVL C01747 V=800.0 PL=0
MOVL C01748 V=800.0 PL=0
MOVL C01749 V=800.0 PL=0
MOVL C01750 V=800.0 PL=0
MOVL C01751 V=800.0 PL=0
MOVL C01752 V=800.0 PL=0
MOVL C01753 V=800.0 PL=0
MOVL C01754 V=800.0 PL=0
MOVL C01755 V=800.0 PL=0
MOVL C01756 V=800.0 PL=0
MOVL C01757 V=800.0 PL=0
MOVL C01758 V=800.0 PL=0
MOVL C01759 V=800.0 PL=0
MOVL C01760 V=800.0 PL=0
MOVL C01761 V=800.0 PL=0
MOVL C01762 V=800.0 PL=0
MOVL C01763 V=800.0 PL=0
MOVL C01764 V=800.0 PL=0
MOVL C01765 V=800.0 PL=0
MOVL C01766 V=800.0 PL=0
MOVL C01767 V=800.0 PL=0
MOVL C01768 V=800.0 PL=0
MOVL C01769 V=800.0 PL=0
MOVL C01770 V=800.0 PL=0
MOVL C01771 V=800.0 PL=0
MOVL C01772 V=800.0 PL=0
MOVL C01773 V=800.0 PL=0
MOVL C01774 V=800.0 PL=0
MOVL C01775 V=800.0 PL=0
MOVL C01776 V=800.0 PL=0
MOVL C01777 V=800.0 PL=0
MOVL C01778 V=800.0 PL=0
MOVL C01779 V=800.0 PL=0
MOVL C01780 V=800.0 PL=0
MOVL C01781 V=800.0 PL=0
MOVL C01782 V=800.0 PL=0
MOVL C01783 V=800.0 PL=0
MOVL C01784 V=800.0 PL=0
MOVL C01785 V=800.0 PL=0
MOVL C01786 V=800.0 PL=0
MOVL C01787 V=800.0 PL=0
MOVL C01788 V=800.0 PL=0
MOVL C01789 V=800.0 PL=0
MOVL C01790 V=800.0 PL=0
MOVL C01791 V=800.0 PL=0
MOVL C01792 V=800.0 PL=0
MOVL C01793 V=800.0 PL=0
MOVL C01794 V=800.0 PL=0
MOVL C01795 V=800.0 PL=0
MOVL C01796 V=800.0 PL=0
MOVL C01797 V=800.0 PL=0
MOVL C01798 V=800.0 PL=0
MOVL C01799 V=800.0 PL=0
MOVL C01800 V=800.0 PL=0
MOVL C01801 V=800.0 PL=0
MOVL C01802 V=800.0 PL=0
MOVL C01803 V=800.0 PL=0
MOVL C01804 V=800.0 PL=0
MOVL C01805 V=800.0 PL=0
MOVL C01806 V=800.0 PL=0
MOVL C01807 V=800.0 PL=0
MOVL C01808 V=800.0 PL=0
MOVL C01809 V=800.0 PL=0
MOVL C01810 V=800.0 PL=0
MOVL C01811 V=800.0 PL=0
MOVL C01812 V=800.0 PL=0
MOVL C01813 V=800.0 PL=0
MOVL C01814 V=800.0 PL=0
MOVL C01815 V=800.0 PL=0
MOVL C01816 V=800.0 PL=0
MOVL C01817 V=800.0 PL=0
MOVL C01818 V=800.0 PL=0
MOVL C01819 V=800.0 PL=0
MOVL C01820 V=800.0 PL=0
MOVL C01821 V=800.0 PL=0
MOVL C01822 V=800.0 PL=0
MOVL C01823 V=800.0 PL=0
MOVL C01824 V=800.0 PL=0
MOVL C01825 V=800.0 PL=0
MOVL C01826 V=800.0 PL=0
MOVL C01827 V=800.0 PL=0
MOVL C01828 V=800.0 PL=0
MOVL C01829 V=800.0 PL=0
MOVL C01830 V=800.0 PL=0
MOVL C01831 V=800.0 PL=0
MOVL C01832 V=800.0 PL=0
MOVL C01833 V=800.0 PL=0
MOVL C01834 V=800.0 PL=0
MOVL C01835 V=800.0 PL=0
MOVL C01836 V=800.0 PL=0
MOVL C01837 V=800.0 PL=0
MOVL C01838 V=800.0 PL=0
MOVL C01839 V=800.0 PL=0
MOVL C01840 V=800.0 PL=0
MOVL C01841 V=800.0 PL=0
MOVL C01842 V=800.0 PL=0
MOVL C01843 V=800.0 PL=0
MOVL C01844 V=800.0 PL=0
MOVL C01845 V=800.0 PL=0
MOVL C01846 V=800.0 PL=0
MOVL C01847 V=800.0 PL=0
MOVL C01848 V=800.0 PL=0
MOVL C01849 V=800.0 PL=0
MOVL C01850 V=800.0 PL=0
MOVL C01851 V=800.0 PL=0
MOVL C01852 V=800.0 PL=0
MOVL C01853 V=800.0 PL=0
MOVL C01854 V=800.0 PL=0
MOVL C01855 V=800.0 PL=0
MOVL C01856 V=800.0 PL=0
MOVL C01857 V=800.0 PL=0
MOVL C01858 V=800.0 PL=0
MOVL C01859 V=800.0 PL=0
MOVL C01860 V=800.0 PL=0
MOVL C01861 V=800.0 PL=0
MOVL C01862 V=800.0 PL=0
MOVL C01863 V=800.0 PL=0
MOVL C01864 V=800.0 PL=0
MOVL C01865 V=800.0 PL=0
MOVL C01866 V=800.0 PL=0
MOVL C01867 V=800.0 PL=0
MOVL C01868 V=800.0 PL=0
MOVL C01869 V=800.0 PL=0
MOVL C01870 V=800.0 PL=0
MOVL C01871 V=800.0 PL=0
MOVL C01872 V=800.0 PL=0
MOVL C01873 V=800.0 PL=0
MOVL C01874 V=800.0 PL=0
MOVL C01875 V=800.0 PL=0
MOVL C01876 V=800.0 PL=0
MOVL C01877 V=800.0 PL=0
MOVL C01878 V=800.0 PL=0
MOVL C01879 V=800.0 PL=0
MOVL C01880 V=800.0 PL=0
MOVL C01881 V=800.0 PL=0
MOVL C01882 V=800.0 PL=0
MOVL C01883 V=800.0 PL=0
MOVL C01884 V=800.0 PL=0
MOVL C01885 V=800.0 PL=0
MOVL C01886 V=800.0 PL=0
MOVL C01887 V=800.0 PL=0
MOVL C01888 V=800.0 PL=0
MOVL C01889 V=800.0 PL=0
MOVL C01890 V=800.0 PL=0
MOVL C01891 V=800.0 PL=0
MOVL C01892 V=800.0 PL=0
MOVL C01893 V=800.0 PL=0
MOVL C01894 V=800.0 PL=0
MOVL C01895 V=800.0 PL=0
MOVL C01896 V=800.0 PL=0
MOVL C01897 V=800.0 PL=0
MOVL C01898 V=800.0 PL=0
MOVL C01899 V=800.0 PL=0
MOVL C01900 V=800.0 PL=0
MOVL C01901 V=800.0 PL=0
MOVL C01902 V=800.0 PL=0
MOVL C01903 V=800.0 PL=0
MOVL C01904 V=800.0 PL=0
MOVL C01905 V=800.0 PL=0
MOVL C01906 V=800.0 PL=0
MOVL C01907 V=800.0 PL=0
MOVL C01908 V=800.0 PL=0
MOVL C01909 V=800.0 PL=0
MOVL C01910 V=800.0 PL=0
MOVL C01911 V=800.0 PL=0
MOVL C01912 V=800.0 PL=0
MOVL C01913 V=800.0 PL=0
MOVL C01914 V=800.0 PL=0
MOVL C01915 V=800.0 PL=0
MOVL C01916 V=800.0 PL=0
MOVL C01917 V=800.0 PL=0
MOVL C01918 V=800.0 PL=0
MOVL C01919 V=800.0 PL=0
MOVL C01920 V=800.0 PL=0
MOVL C01921 V=800.0 PL=0
MOVL C01922 V=800.0 PL=0
MOVL C01923 V=800.0 PL=0
MOVL C01924 V=800.0 PL=0
MOVL C01925 V=800.0 PL=0
MOVL C01926 V=800.0 PL=0
